# B&R Automation Studio project NAELD004C00R10L518F00 (part 19)

#### Act_OptP1031LifterMask.st
```iecst
ACTION Act_OptP1031LifterMask:

	// Interlock Power
	IF p_bLifterBtmAxisErr = TRUE AND p_bLifterBtmPwrOn = FALSE THEN
		fUIInRtStatOff(ADR(tyP1031MagSetTeach.tyMotionStdLifter.tyBtnPwr.uiMaskRtStat));
		tyP1031MagSetTeach.tyMotionStdLifter.tyBtnPwr.bValue		:= FALSE;
	ELSE
		fUIInRtStatHide(ADR(tyP1031MagSetTeach.tyMotionStdLifter.tyBtnPwr.uiMaskRtStat));
	END_IF

	// Interlock Others Move
	IF p_bLifterBtmAxisErr = TRUE OR p_bLifterBtmPwrOn = FALSE THEN
		fUIInRtStatOff(ADR(tyP1031MagSetTeach.tyMotionStdLifter.tyBtnOrigin.uiMaskRtStat));
		fUIInRtStatOff(ADR(tyP1031MagSetTeach.tyMotionStdLifter.tyBtnMovRel.uiMaskRtStat));
		fUIInRtStatOff(ADR(tyP1031MagSetTeach.tyMotionStdLifter.tyBtnJogUp.uiMaskRtStat));
		fUIInRtStatOff(ADR(tyP1031MagSetTeach.tyMotionStdLifter.tyBtnJogDown.uiMaskRtStat));
	ELSE
		fUIInRtStatHide(ADR(tyP1031MagSetTeach.tyMotionStdLifter.tyBtnOrigin.uiMaskRtStat));
		fUIInRtStatHide(ADR(tyP1031MagSetTeach.tyMotionStdLifter.tyBtnMovRel.uiMaskRtStat));
		fUIInRtStatHide(ADR(tyP1031MagSetTeach.tyMotionStdLifter.tyBtnJogUp.uiMaskRtStat));
		fUIInRtStatHide(ADR(tyP1031MagSetTeach.tyMotionStdLifter.tyBtnJogDown.uiMaskRtStat));
	END_IF

	// Interlock Move Absolute
	IF p_bLifterBtmAxisErr = TRUE OR p_bLifterBtmPwrOn = FALSE OR p_bLifterBtmIsHomed = FALSE THEN

		fUIInRtStatOff(ADR(tyP1031MagSetTeach.tyTeachLifterMag1Slt1Pos.tyBtn2.uiMaskRtStat));
		fUIInRtStatOff(ADR(tyP1031MagSetTeach.tyTeachLifterMag2Slt1Pos.tyBtn2.uiMaskRtStat));
		fUIInRtStatOff(ADR(tyP1031MagSetTeach.tyTeachLifterMag3Slt1Pos.tyBtn2.uiMaskRtStat));
		fUIInRtStatOff(ADR(tyP1031MagSetTeach.tyTeachLifterMag4Slt1Pos.tyBtn2.uiMaskRtStat));
		fUIInRtStatOff(ADR(tyP1031MagSetTeach.tyMotionStdLifter.tyBtnMovAbs.uiMaskRtStat));
	ELSE
		fUIInRtStatHide(ADR(tyP1031MagSetTeach.tyTeachLifterMag1Slt1Pos.tyBtn2.uiMaskRtStat));
		fUIInRtStatHide(ADR(tyP1031MagSetTeach.tyTeachLifterMag2Slt1Pos.tyBtn2.uiMaskRtStat));
		fUIInRtStatHide(ADR(tyP1031MagSetTeach.tyTeachLifterMag3Slt1Pos.tyBtn2.uiMaskRtStat));
		fUIInRtStatHide(ADR(tyP1031MagSetTeach.tyTeachLifterMag4Slt1Pos.tyBtn2.uiMaskRtStat));
		fUIInRtStatHide(ADR(tyP1031MagSetTeach.tyMotionStdLifter.tyBtnMovAbs.uiMaskRtStat));
	END_IF

	//Interlock Limit Sensor
	IF tyP1031MagSetTeach.tyMotionStdLifter.tyBtnDownLmtSen.bValue = TRUE THEN
		fUIInRtStatOff(ADR(tyP1031MagSetTeach.tyMotionStdLifter.tyBtnJogDown.uiMaskRtStat));
	END_IF

	IF tyP1031MagSetTeach.tyMotionStdLifter.tyBtnUpLmtSen.bValue = TRUE THEN
		fUIInRtStatOff(ADR(tyP1031MagSetTeach.tyMotionStdLifter.tyBtnJogUp.uiMaskRtStat));
	END_IF

	// Interlock When Moving
	IF tyP1031MagSetTeach.tyMotionStdLifter.tyBtnOrigin.bRtCompl = TRUE THEN
		fUIInRtStatOff(ADR(tyP1031MagSetTeach.tyMotionStdLifter.tyBtnMovAbs.uiMaskRtStat));
		fUIInRtStatOff(ADR(tyP1031MagSetTeach.tyMotionStdLifter.tyBtnMovRel.uiMaskRtStat));
		fUIInRtStatOff(ADR(tyP1031MagSetTeach.tyMotionStdLifter.tyBtnJogUp.uiMaskRtStat));
		fUIInRtStatOff(ADR(tyP1031MagSetTeach.tyMotionStdLifter.tyBtnJogDown.uiMaskRtStat));

		fUIInRtStatOff(ADR(tyP1031MagSetTeach.tyTeachLifterMag1Slt1Pos.tyBtn2.uiMaskRtStat));
		fUIInRtStatOff(ADR(tyP1031MagSetTeach.tyTeachLifterMag2Slt1Pos.tyBtn2.uiMaskRtStat));
		fUIInRtStatOff(ADR(tyP1031MagSetTeach.tyTeachLifterMag3Slt1Pos.tyBtn2.uiMaskRtStat));
		fUIInRtStatOff(ADR(tyP1031MagSetTeach.tyTeachLifterMag4Slt1Pos.tyBtn2.uiMaskRtStat));

	ELSIF tyP1031MagSetTeach.tyMotionStdLifter.tyBtnMovAbs.bRtCompl = TRUE THEN
		fUIInRtStatOff(ADR(tyP1031MagSetTeach.tyMotionStdLifter.tyBtnOrigin.uiMaskRtStat));
		fUIInRtStatOff(ADR(tyP1031MagSetTeach.tyMotionStdLifter.tyBtnMovRel.uiMaskRtStat));
		fUIInRtStatOff(ADR(tyP1031MagSetTeach.tyMotionStdLifter.tyBtnJogUp.uiMaskRtStat));
		fUIInRtStatOff(ADR(tyP1031MagSetTeach.tyMotionStdLifter.tyBtnJogDown.uiMaskRtStat));

		fUIInRtStatOff(ADR(tyP1031MagSetTeach.tyTeachLifterMag1Slt1Pos.tyBtn2.uiMaskRtStat));
		fUIInRtStatOff(ADR(tyP1031MagSetTeach.tyTeachLifterMag2Slt1Pos.tyBtn2.uiMaskRtStat));
		fUIInRtStatOff(ADR(tyP1031MagSetTeach.tyTeachLifterMag3Slt1Pos.tyBtn2.uiMaskRtStat));
		fUIInRtStatOff(ADR(tyP1031MagSetTeach.tyTeachLifterMag4Slt1Pos.tyBtn2.uiMaskRtStat));

	ELSIF tyP1031MagSetTeach.tyMotionStdLifter.tyBtnMovRel.bRtCompl = TRUE THEN
		fUIInRtStatOff(ADR(tyP1031MagSetTeach.tyMotionStdLifter.tyBtnOrigin.uiMaskRtStat));
		fUIInRtStatOff(ADR(tyP1031MagSetTeach.tyMotionStdLifter.tyBtnMovAbs.uiMaskRtStat));
		fUIInRtStatOff(ADR(tyP1031MagSetTeach.tyMotionStdLifter.tyBtnJogUp.uiMaskRtStat));
		fUIInRtStatOff(ADR(tyP1031MagSetTeach.tyMotionStdLifter.tyBtnJogDown.uiMaskRtStat));

		fUIInRtStatOff(ADR(tyP1031MagSetTeach.tyTeachLifterMag1Slt1Pos.tyBtn2.uiMaskRtStat));
		fUIInRtStatOff(ADR(tyP1031MagSetTeach.tyTeachLifterMag2Slt1Pos.tyBtn2.uiMaskRtStat));
		fUIInRtStatOff(ADR(tyP1031MagSetTeach.tyTeachLifterMag3Slt1Pos.tyBtn2.uiMaskRtStat));
		fUIInRtStatOff(ADR(tyP1031MagSetTeach.tyTeachLifterMag4Slt1Pos.tyBtn2.uiMaskRtStat));

	ELSIF tyP1031MagSetTeach.tyMotionStdLifter.tyBtnJogDown.bRtCompl = TRUE OR tyP1031MagSetTeach.tyMotionStdLifter.tyBtnJogDown.bValue = TRUE THEN
		fUIInRtStatOff(ADR(tyP1031MagSetTeach.tyMotionStdLifter.tyBtnOrigin.uiMaskRtStat));
		fUIInRtStatOff(ADR(tyP1031MagSetTeach.tyMotionStdLifter.tyBtnMovAbs.uiMaskRtStat));
		fUIInRtStatOff(ADR(tyP1031MagSetTeach.tyMotionStdLifter.tyBtnMovRel.uiMaskRtStat));
		fUIInRtStatOff(ADR(tyP1031MagSetTeach.tyMotionStdLifter.tyBtnJogUp.uiMaskRtStat));

		fUIInRtStatOff(ADR(tyP1031MagSetTeach.tyTeachLifterMag1Slt1Pos.tyBtn2.uiMaskRtStat));
		fUIInRtStatOff(ADR(tyP1031MagSetTeach.tyTeachLifterMag2Slt1Pos.tyBtn2.uiMaskRtStat));
		fUIInRtStatOff(ADR(tyP1031MagSetTeach.tyTeachLifterMag3Slt1Pos.tyBtn2.uiMaskRtStat));
		fUIInRtStatOff(ADR(tyP1031MagSetTeach.tyTeachLifterMag4Slt1Pos.tyBtn2.uiMaskRtStat));

	ELSIF tyP1031MagSetTeach.tyMotionStdLifter.tyBtnJogUp.bRtCompl = TRUE OR tyP1031MagSetTeach.tyMotionStdLifter.tyBtnJogUp.bValue = TRUE THEN
		fUIInRtStatOff(ADR(tyP1031MagSetTeach.tyMotionStdLifter.tyBtnOrigin.uiMaskRtStat));
		fUIInRtStatOff(ADR(tyP1031MagSetTeach.tyMotionStdLifter.tyBtnMovAbs.uiMaskRtStat));
		fUIInRtStatOff(ADR(tyP1031MagSetTeach.tyMotionStdLifter.tyBtnMovRel.uiMaskRtStat));
		fUIInRtStatOff(ADR(tyP1031MagSetTeach.tyMotionStdLifter.tyBtnJogDown.uiMaskRtStat));

		fUIInRtStatOff(ADR(tyP1031MagSetTeach.tyTeachLifterMag1Slt1Pos.tyBtn2.uiMaskRtStat));
		fUIInRtStatOff(ADR(tyP1031MagSetTeach.tyTeachLifterMag2Slt1Pos.tyBtn2.uiMaskRtStat));
		fUIInRtStatOff(ADR(tyP1031MagSetTeach.tyTeachLifterMag3Slt1Pos.tyBtn2.uiMaskRtStat));
		fUIInRtStatOff(ADR(tyP1031MagSetTeach.tyTeachLifterMag4Slt1Pos.tyBtn2.uiMaskRtStat));

	ELSIF tyP1031MagSetTeach.tyTeachLifterMag1Slt1Pos.tyBtn2.bRtCompl = TRUE THEN
		fUIInRtStatOff(ADR(tyP1031MagSetTeach.tyMotionStdLifter.tyBtnOrigin.uiMaskRtStat));
		fUIInRtStatOff(ADR(tyP1031MagSetTeach.tyMotionStdLifter.tyBtnMovAbs.uiMaskRtStat));
		fUIInRtStatOff(ADR(tyP1031MagSetTeach.tyMotionStdLifter.tyBtnMovRel.uiMaskRtStat));
		fUIInRtStatOff(ADR(tyP1031MagSetTeach.tyMotionStdLifter.tyBtnJogUp.uiMaskRtStat));
		fUIInRtStatOff(ADR(tyP1031MagSetTeach.tyMotionStdLifter.tyBtnJogDown.uiMaskRtStat));

	ELSIF tyP1031MagSetTeach.tyTeachLifterMag2Slt1Pos.tyBtn2.bRtCompl = TRUE THEN
		fUIInRtStatOff(ADR(tyP1031MagSetTeach.tyMotionStdLifter.tyBtnOrigin.uiMaskRtStat));
		fUIInRtStatOff(ADR(tyP1031MagSetTeach.tyMotionStdLifter.tyBtnMovAbs.uiMaskRtStat));
		fUIInRtStatOff(ADR(tyP1031MagSetTeach.tyMotionStdLifter.tyBtnMovRel.uiMaskRtStat));
		fUIInRtStatOff(ADR(tyP1031MagSetTeach.tyMotionStdLifter.tyBtnJogUp.uiMaskRtStat));
		fUIInRtStatOff(ADR(tyP1031MagSetTeach.tyMotionStdLifter.tyBtnJogDown.uiMaskRtStat));

	ELSIF tyP1031MagSetTeach.tyTeachLifterMag3Slt1Pos.tyBtn2.bRtCompl = TRUE THEN
		fUIInRtStatOff(ADR(tyP1031MagSetTeach.tyMotionStdLifter.tyBtnOrigin.uiMaskRtStat));
		fUIInRtStatOff(ADR(tyP1031MagSetTeach.tyMotionStdLifter.tyBtnMovAbs.uiMaskRtStat));
		fUIInRtStatOff(ADR(tyP1031MagSetTeach.tyMotionStdLifter.tyBtnMovRel.uiMaskRtStat));
		fUIInRtStatOff(ADR(tyP1031MagSetTeach.tyMotionStdLifter.tyBtnJogUp.uiMaskRtStat));
		fUIInRtStatOff(ADR(tyP1031MagSetTeach.tyMotionStdLifter.tyBtnJogDown.uiMaskRtStat));

	END_IF

	//Axis Error
	IF tyP1031MagSetTeach.tyMotionStdLifter.tyBtnPwr.bRtCompl = TRUE THEN
		fUIInRtStatOff(ADR(tyP1031MagSetTeach.tyMotionStdLifter.tyBtnRst.uiMaskRtStat));
	ELSE
		fUIInRtStatHide(ADR(tyP1031MagSetTeach.tyMotionStdLifter.tyBtnRst.uiMaskRtStat));
	END_IF

	//Interlock Button Get
	IF p_bLifterBtmAxisErr = TRUE OR p_bLifterBtmIsHomed = FALSE OR p_bLifterBtmFwdLmtSen = TRUE OR p_bLifterBtmRevLmtSen = TRUE THEN
		fUIInRtStatOff(ADR(tyP1031MagSetTeach.tyTeachLifterMag1Slt1Pos.tyBtn1.uiMaskRtStat));
		fUIInRtStatOff(ADR(tyP1031MagSetTeach.tyTeachLifterMag2Slt1Pos.tyBtn1.uiMaskRtStat));
		fUIInRtStatOff(ADR(tyP1031MagSetTeach.tyTeachLifterMag3Slt1Pos.tyBtn1.uiMaskRtStat));
		fUIInRtStatOff(ADR(tyP1031MagSetTeach.tyTeachLifterMag4Slt1Pos.tyBtn1.uiMaskRtStat));
	ELSE
		fUIInRtStatHide(ADR(tyP1031MagSetTeach.tyTeachLifterMag1Slt1Pos.tyBtn1.uiMaskRtStat));
		fUIInRtStatHide(ADR(tyP1031MagSetTeach.tyTeachLifterMag2Slt1Pos.tyBtn1.uiMaskRtStat));
		fUIInRtStatHide(ADR(tyP1031MagSetTeach.tyTeachLifterMag3Slt1Pos.tyBtn1.uiMaskRtStat));
		fUIInRtStatHide(ADR(tyP1031MagSetTeach.tyTeachLifterMag4Slt1Pos.tyBtn1.uiMaskRtStat));
	END_IF

END_ACTION
```

#### Act_OptP1031LifterUpdtDat.st
```iecst
ACTION Act_OptP1031LifterUpdtDat:

	tyP1031MagSetTeach.tyMotionStdLifter.tyNumCurrPos.diValue		:= p_diLifterBtmActualPos;
	tyP1031MagSetTeach.tyMotionStdLifter.tyNumErrCode.diValue		:= UDINT_TO_DINT(p_udiLifterBtmAxisErrID);
	tyP1031MagSetTeach.tyMotionStdLifter.tyBitmapPwr.usiValueIdx	:= BOOL_TO_USINT(p_bLifterBtmPwrOn);
	tyP1031MagSetTeach.tyMotionStdLifter.tyBitmapRst.usiValueIdx	:= BOOL_TO_USINT(NOT p_bLifterBtmAxisErr);
	tyP1031MagSetTeach.tyMotionStdLifter.tyBitmapOrigin.usiValueIdx	:= BOOL_TO_USINT(p_bLifterBtmIsHomed);
	tyP1031MagSetTeach.tyMotionStdLifter.tyBtnUpLmtSen.bValue		:= p_bLifterBtmUpSen;
	tyP1031MagSetTeach.tyMotionStdLifter.tyBtnDownLmtSen.bValue		:= p_bLifterBtmDownSen;

	//Machine Bitmap
	IF   (p_tyNtParamCurr.eProjMag = LDMagDual AND p_tyNtParamCurr.bMagAutoVerifyPrep = FALSE)
		OR (p_tyNtParamCurr.eProjMag = LDMagTriple AND p_tyNtParamCurr.bMagAutoVerifyPrep = FALSE)
		OR (p_tyNtParamCurr.eProjMag = LDMagDual AND p_tyNtParamCurr.bMagAutoVerifyPrep = TRUE)
		THEN
		IF p_bLifterBtmIsHomed = TRUE THEN

			IF p_diLifterBtmActualPos <= (p_tyNtParamCurr.tyUILifterTargetPos.diMax / 3) THEN
				tyP1031MagSetTeach.tyMotionStdLifter.tyBitmapMc.uiValueIdx 	:= 2;
			ELSIF p_diLifterBtmActualPos <= (p_tyNtParamCurr.tyUILifterTargetPos.diMax / 3 * 2) THEN
				tyP1031MagSetTeach.tyMotionStdLifter.tyBitmapMc.uiValueIdx 	:= 3;
			ELSE
				tyP1031MagSetTeach.tyMotionStdLifter.tyBitmapMc.uiValueIdx 	:= 4;
			END_IF

		ELSE
			tyP1031MagSetTeach.tyMotionStdLifter.tyBitmapMc.uiValueIdx	:= 2;
		END_IF

	ELSIF p_tyNtParamCurr.eProjMag = LDMagTriple AND p_tyNtParamCurr.bMagAutoVerifyPrep = TRUE
		THEN
		IF p_bLifterBtmIsHomed = TRUE THEN

			IF p_diLifterBtmActualPos <= (p_tyNtParamCurr.tyUILifterTargetPos.diMax / 3) THEN
				tyP1031MagSetTeach.tyMotionStdLifter.tyBitmapMc.uiValueIdx 	:= 23;
			ELSIF p_diLifterBtmActualPos <= (p_tyNtParamCurr.tyUILifterTargetPos.diMax / 3 * 2) THEN
				tyP1031MagSetTeach.tyMotionStdLifter.tyBitmapMc.uiValueIdx 	:= 24;
			ELSE
				tyP1031MagSetTeach.tyMotionStdLifter.tyBitmapMc.uiValueIdx 	:= 25;
			END_IF

		ELSE
			tyP1031MagSetTeach.tyMotionStdLifter.tyBitmapMc.uiValueIdx	:= 23;
		END_IF

	ELSIF p_tyNtParamCurr.eProjMag = LDMagQuadruple AND p_tyNtParamCurr.bMagAutoVerifyPrep = TRUE
		THEN
		IF p_bLifterBtmIsHomed = TRUE THEN

			IF p_diLifterBtmActualPos <= (p_tyNtParamCurr.tyUILifterTargetPos.diMax / 3) THEN
				tyP1031MagSetTeach.tyMotionStdLifter.tyBitmapMc.uiValueIdx 	:= 27;
			ELSIF p_diLifterBtmActualPos <= (p_tyNtParamCurr.tyUILifterTargetPos.diMax / 3 * 2) THEN
				tyP1031MagSetTeach.tyMotionStdLifter.tyBitmapMc.uiValueIdx 	:= 28;
			ELSE
				tyP1031MagSetTeach.tyMotionStdLifter.tyBitmapMc.uiValueIdx 	:= 29;
			END_IF

		ELSE
			tyP1031MagSetTeach.tyMotionStdLifter.tyBitmapMc.uiValueIdx	:= 27;
		END_IF
	END_IF

	IF p_tyNtParamCurr.eProjMag = LDMagTriple AND p_tyNtParamCurr.bProjLifterMagPlatform THEN
		IF 	tyP1031MagSetTeach.tyMotionStdLifter.tyBitmapMc.uiValueIdx < 400 THEN
			tyP1031MagSetTeach.tyMotionStdLifter.tyBitmapMc.uiValueIdx	:= tyP1031MagSetTeach.tyMotionStdLifter.tyBitmapMc.uiValueIdx + 400;
		END_IF
	ELSIF (p_tyNtParamCurr.eProjMag = LDMagDual OR p_tyNtParamCurr.eProjMag = LDMagTriple) AND p_tyNtParamCurr.bProjMotorizedPullerPrep = FALSE THEN
		IF 	tyP1031MagSetTeach.tyMotionStdLifter.tyBitmapMc.uiValueIdx < 200 THEN
			tyP1031MagSetTeach.tyMotionStdLifter.tyBitmapMc.uiValueIdx	:= tyP1031MagSetTeach.tyMotionStdLifter.tyBitmapMc.uiValueIdx + 200;
		END_IF
	ELSIF p_tyNtParamCurr.eProjMag = LDMagDual AND p_tyNtParamCurr.bProjMotorizedPullerPrep THEN
		IF p_tyNtParamCurr.sJobNo = '2023-0258A01' THEN
			tyP1031MagSetTeach.tyMotionStdLifter.tyBitmapMc.uiValueIdx	:= tyP1031MagSetTeach.tyMotionStdLifter.tyBitmapMc.uiValueIdx + 444-2;
		END_IF
	ELSIF p_tyNtParamCurr.eProjMag = LDMagTriple AND p_tyNtParamCurr.bMagAutoVerifyPrep = FALSE AND p_tyNtParamCurr.bProjMotorizedPullerPrep = TRUE
		THEN
		IF 	tyP1031MagSetTeach.tyMotionStdLifter.tyBitmapMc.uiValueIdx < 300 THEN
			tyP1031MagSetTeach.tyMotionStdLifter.tyBitmapMc.uiValueIdx	:= tyP1031MagSetTeach.tyMotionStdLifter.tyBitmapMc.uiValueIdx + 300;
		END_IF
	END_IF

END_ACTION
```

#### Act_OptP1031LifterKeypad.st
```iecst
ACTION Act_OptP1031LifterKeypad:

	IF fUIOutRtStatTPIsOpen(ADR(tyP1031MagSetTeach.tyMotionStdLifter.tyNumTargetPos.uiRtStat)) = TRUE THEN
		tyProperty.tyKeypad.tyStringTitle.sKeypadTitle		:= tyP1031MagSetTeach.tyMotionStdLifter.tyNumTargetPos.sKeypadTitle;

	ELSIF fUIOutRtStatTPIsOpen(ADR(tyP1026McSetTeach.tyMotionStdLifter.tyNumStepSize.uiRtStat)) = TRUE THEN
		tyProperty.tyKeypad.tyStringTitle.sKeypadTitle		:= tyP1031MagSetTeach.tyMotionStdLifter.tyNumStepSize.sKeypadTitle;

	ELSIF fUIOutRtStatTPIsOpen(ADR(tyP1031MagSetTeach.tyMotionStdLifter.tyNumNomSpd.uiRtStat)) = TRUE THEN
		tyProperty.tyKeypad.tyStringTitle.sKeypadTitle		:= tyP1031MagSetTeach.tyMotionStdLifter.tyNumNomSpd.sKeypadTitle;

	ELSIF fUIOutRtStatTPIsOpen(ADR(tyP1031MagSetTeach.tyMotionStdLifter.tyNumSlwSpd.uiRtStat)) = TRUE THEN
		tyProperty.tyKeypad.tyStringTitle.sKeypadTitle		:= tyP1031MagSetTeach.tyMotionStdLifter.tyNumSlwSpd.sKeypadTitle;

	ELSIF fUIOutRtStatTPIsOpen(ADR(tyP1031MagSetTeach.tyTeachLifterMag1Slt1Pos.tyNumNewSlt.uiRtStat)) = TRUE THEN
		tyProperty.tyKeypad.tyStringTitle.sKeypadTitle		:= tyP1031MagSetTeach.tyTeachLifterMag1Slt1Pos.tyNumNewSlt.sKeypadTitle;

	ELSIF fUIOutRtStatTPIsOpen(ADR(tyP1031MagSetTeach.tyTeachLifterMag2Slt1Pos.tyNumNewSlt.uiRtStat)) = TRUE THEN
		tyProperty.tyKeypad.tyStringTitle.sKeypadTitle		:= tyP1031MagSetTeach.tyTeachLifterMag2Slt1Pos.tyNumNewSlt.sKeypadTitle;

	ELSIF fUIOutRtStatTPIsOpen(ADR(tyP1031MagSetTeach.tyTeachLifterMag3Slt1Pos.tyNumNewSlt.uiRtStat)) = TRUE THEN
		tyProperty.tyKeypad.tyStringTitle.sKeypadTitle		:= tyP1031MagSetTeach.tyTeachLifterMag3Slt1Pos.tyNumNewSlt.sKeypadTitle;

	ELSIF fUIOutRtStatTPIsOpen(ADR(tyP1031MagSetTeach.tyTeachLifterMag4Slt1Pos.tyNumNewSlt.uiRtStat)) = TRUE THEN
		tyProperty.tyKeypad.tyStringTitle.sKeypadTitle		:= tyP1031MagSetTeach.tyTeachLifterMag4Slt1Pos.tyNumNewSlt.sKeypadTitle;

	END_IF

END_ACTION
```

#### Act_OptP1031LifterRstMnl.st
```iecst
ACTION Act_OptP1031LifterRstMnl:

	IF EDGEPOS((bManualMod = FALSE) OR (p_eLifterBtmStatus = Error)) THEN

		bJogSlow				:= FALSE;
		bJogFast				:= FALSE;
		fbJogSlowToFastDlyTm.IN	:= FALSE;

		tyP1031MagSetTeach.tyMotionStdLifter.tyBtnPwr.bRtCompl			:= FALSE;
		tyP1031MagSetTeach.tyMotionStdLifter.tyBtnStop.bRtCompl			:= FALSE;
		tyP1031MagSetTeach.tyMotionStdLifter.tyBtnOrigin.bRtCompl		:= FALSE;
		tyP1031MagSetTeach.tyMotionStdLifter.tyBtnRst.bRtCompl			:= FALSE;
		tyP1031MagSetTeach.tyMotionStdLifter.tyBtnMovAbs.bRtCompl		:= FALSE;
		tyP1031MagSetTeach.tyMotionStdLifter.tyBtnMovRel.bRtCompl		:= FALSE;
		tyP1031MagSetTeach.tyMotionStdLifter.tyBtnJogUp.bRtCompl		:= FALSE;
		tyP1031MagSetTeach.tyMotionStdLifter.tyBtnJogDown.bRtCompl		:= FALSE;

		tyP1031MagSetTeach.tyTeachLifterMag1Slt1Pos.tyBtn2.bRtCompl		:= FALSE;
		tyP1031MagSetTeach.tyTeachLifterMag2Slt1Pos.tyBtn2.bRtCompl		:= FALSE;
		tyP1031MagSetTeach.tyTeachLifterMag3Slt1Pos.tyBtn2.bRtCompl		:= FALSE;
		tyP1031MagSetTeach.tyTeachLifterMag4Slt1Pos.tyBtn2.bRtCompl		:= FALSE;

		tyP1031MagSetTeach.tyMotionStdLifter.tyBtnPwr.bValue			:= FALSE;
		tyP1031MagSetTeach.tyMotionStdLifter.tyBtnStop.bValue			:= TRUE;
		tyP1031MagSetTeach.tyMotionStdLifter.tyBtnOrigin.bValue			:= FALSE;
		tyP1031MagSetTeach.tyMotionStdLifter.tyBtnRst.bValue			:= FALSE;
		tyP1031MagSetTeach.tyMotionStdLifter.tyBtnMovAbs.bValue			:= FALSE;
		tyP1031MagSetTeach.tyMotionStdLifter.tyBtnMovRel.bValue			:= FALSE;
		tyP1031MagSetTeach.tyMotionStdLifter.tyBtnJogUp.bValue			:= FALSE;
		tyP1031MagSetTeach.tyMotionStdLifter.tyBtnJogDown.bValue		:= FALSE;

		tyP1031MagSetTeach.tyTeachLifterMag1Slt1Pos.tyBtn2.bValue		:= FALSE;
		tyP1031MagSetTeach.tyTeachLifterMag2Slt1Pos.tyBtn2.bValue		:= FALSE;
		tyP1031MagSetTeach.tyTeachLifterMag3Slt1Pos.tyBtn2.bValue		:= FALSE;
		tyP1031MagSetTeach.tyTeachLifterMag4Slt1Pos.tyBtn2.bValue		:= FALSE;

		tyP1031MagSetTeach.tyMotionStdLifter.tyBtnPwr.bRtLk				:= FALSE;
		tyP1031MagSetTeach.tyMotionStdLifter.tyBtnStop.bRtLk			:= TRUE;
		tyP1031MagSetTeach.tyMotionStdLifter.tyBtnOrigin.bRtLk			:= FALSE;
		tyP1031MagSetTeach.tyMotionStdLifter.tyBtnRst.bRtLk				:= FALSE;
		tyP1031MagSetTeach.tyMotionStdLifter.tyBtnMovAbs.bRtLk			:= FALSE;
		tyP1031MagSetTeach.tyMotionStdLifter.tyBtnMovRel.bRtLk			:= FALSE;
		tyP1031MagSetTeach.tyMotionStdLifter.tyBtnJogUp.bRtLk			:= FALSE;
		tyP1031MagSetTeach.tyMotionStdLifter.tyBtnJogDown.bRtLk			:= FALSE;

		tyP1031MagSetTeach.tyTeachLifterMag1Slt1Pos.tyBtn2.bRtLk		:= FALSE;
		tyP1031MagSetTeach.tyTeachLifterMag2Slt1Pos.tyBtn2.bRtLk		:= FALSE;
		tyP1031MagSetTeach.tyTeachLifterMag3Slt1Pos.tyBtn2.bRtLk		:= FALSE;
		tyP1031MagSetTeach.tyTeachLifterMag4Slt1Pos.tyBtn2.bRtLk		:= FALSE;

		tyP1031MagSetTeach.tyMotionStdLifter.tyBtnPwr.uiMaskRtStat		:= TRUE;
		tyP1031MagSetTeach.tyMotionStdLifter.tyBtnOrigin.uiMaskRtStat	:= FALSE;
		tyP1031MagSetTeach.tyMotionStdLifter.tyBtnRst.uiMaskRtStat		:= TRUE;
		tyP1031MagSetTeach.tyMotionStdLifter.tyBtnMovAbs.uiMaskRtStat	:= FALSE;
		tyP1031MagSetTeach.tyMotionStdLifter.tyBtnMovRel.uiMaskRtStat	:= FALSE;
		tyP1031MagSetTeach.tyMotionStdLifter.tyBtnJogUp.uiMaskRtStat	:= FALSE;
		tyP1031MagSetTeach.tyMotionStdLifter.tyBtnJogDown.uiMaskRtStat	:= FALSE;

		tyP1031MagSetTeach.tyTeachLifterMag1Slt1Pos.tyBtn2.uiMaskRtStat	:= FALSE;
		tyP1031MagSetTeach.tyTeachLifterMag2Slt1Pos.tyBtn2.uiMaskRtStat	:= FALSE;
		tyP1031MagSetTeach.tyTeachLifterMag3Slt1Pos.tyBtn2.uiMaskRtStat	:= FALSE;
		tyP1031MagSetTeach.tyTeachLifterMag4Slt1Pos.tyBtn2.uiMaskRtStat	:= FALSE;

		eInShutterAct	:= PneuActIdle;
		eOutShutterAct	:= PneuActIdle;
		eLifterBtmAct	:= LifterActIdle;

		tyP1031MagSetTeach.tyInOutletShutterFB.tyBtnClose.bRtCompl	:= FALSE;
		tyP1031MagSetTeach.tyInOutletShutterFB.tyBtnClose.bValue	:= FALSE;
		tyP1031MagSetTeach.tyInOutletShutterFB.tyBtnOpen.bRtCompl	:= FALSE;
		tyP1031MagSetTeach.tyInOutletShutterFB.tyBtnOpen.bValue	:= FALSE;
	END_IF

END_ACTION
```

#### Act_EntP1040Disp.st
```iecst
ACTION Act_EntP1040Disp:

	//Access Address
	p_tyC0005Main ACCESS ADR(tyCommon.tyMain);

	p_tyC0007Notif ACCESS ADR(tyCommon.tyNotif);

	p_tyC0008MsgBox ACCESS ADR(tyP1040ProdSet.tyMsgBoxHide);

	p_tyC0009Info ACCESS ADR(tyCommon.tyInfo);

	p_tyC0011RcpPopUp ACCESS ADR(tyP1040ProdSet.tyRcpPopUp);

	p_tyP1040ProdSet ACCESS ADR(tyP1040ProdSet.tyProdSet);
	tyP1040ProdSet.tyProdSet.tyStringSearch.sValue					:= '';

	//Display
	udiP1040SelectedRowOld	:= 0;

	tyP1040ProdSet.tyProdSet.tyBtnLongBrd.uiRtStat.0	:= NOT(p_tyNtParamCurr.bProjLongBrdPrep AND p_tyMcParamCurr.bLongBrdEn);

	//tyP1040ProdSet.tyProdSet.tyNumLastSlt.diValueMax	:= p_tyMagRcpCurrRcp.diTtlSlt;
	tyP1040ProdSet.tyProdSet.tyNumLastSlt.diValueMax	:= p_tyNtParamCurr.tyProdRcpMaxSlt.diMax;
	tyP1040ProdSet.tyProdSet.tyNumLastSltRear.diValueMax	:= p_tyMagRcpCurrRcp.diTtlSlt;

	fUIInRtStatHide(ADR(tyP1040ProdSet.tyRcpPopUp.tyLyr.uiRtStat));

END_ACTION
```

#### Act_OptP1040Del.st
```iecst
ACTION Act_OptP1040Del:

	IF tyP1040ProdSet.tyProdSet.tyBtnDelete.bRtCompl = TRUE THEN
		IF usiDelProdRcpStep = 0 THEN
			tyP1040ProdSet.tyProdSet.tyStringSearch.uiMaskRtStat				:= FALSE;
			tyP1040ProdSet.tyProdSet.tyTableRecipe.uiMaskRtStat					:= FALSE;

			IF tyP1040ProdSet.tyProdSet.tyTableRecipe.a_tyStringDataCol1[tyP1040Table.uiSelectedRow].sValue = p_tyProdRcpCurrRcp0.sRcpNm THEN
				p_tyC0008MsgBox ACCESS ADR(tyP1040ProdSet.tyMsgBoxDelCurrRcpAsk);

				IF tyP1040ProdSet.tyMsgBoxDelCurrRcpAsk.tyBtnNo.bRtCompl = TRUE THEN
					tyP1040ProdSet.tyMsgBoxDelCurrRcpAsk.tyBtnNo.bRtCompl 		:= FALSE;
					tyP1040ProdSet.tyMsgBoxDelCurrRcpAsk.tyBtnNo.bValue 		:= FALSE;

					p_tyC0008MsgBox ACCESS ADR(tyP1040ProdSet.tyMsgBoxHide);

					usiDelProdRcpStep	:= 99;
				END_IF
			ELSE
				p_tyC0008MsgBox ACCESS ADR(tyP1040ProdSet.tyMsgBoxDelAsk);

				IF tyP1040ProdSet.tyMsgBoxDelAsk.tyBtnYes.bRtCompl = TRUE THEN
					tyP1040ProdSet.tyMsgBoxDelAsk.tyBtnYes.bRtCompl				:= FALSE;
					tyP1040ProdSet.tyMsgBoxDelAsk.tyBtnYes.bValue				:= FALSE;

					p_tyC0008MsgBox ACCESS ADR(tyP1040ProdSet.tyMsgBoxHide);

					usiDelProdRcpStep	:= 1;

				ELSIF tyP1040ProdSet.tyMsgBoxDelAsk.tyBtnNo.bRtCompl = TRUE THEN
					tyP1040ProdSet.tyMsgBoxDelAsk.tyBtnNo.bRtCompl				:= FALSE;
					tyP1040ProdSet.tyMsgBoxDelAsk.tyBtnNo.bValue				:= FALSE;

					p_tyC0008MsgBox ACCESS ADR(tyP1040ProdSet.tyMsgBoxHide);

					usiDelProdRcpStep	:= 99;

				END_IF
			END_IF

		ELSIF usiDelProdRcpStep = 1 THEN
			tyProdRcpInfoIn.sRcpNm			:= tyP1040ProdSet.tyProdSet.tyTableRecipe.a_tyStringDataCol1[tyP1040Table.uiSelectedRow].sValue;

			eProdRcpAct					:= ProdRcpActDel;

			IF p_eProdRcpStat = ProdRcpActDel AND p_eProdRcpStatus = Done THEN
				eProdRcpAct				:= ProdRcpActIdle;

				IF p_bProdRcpNmEmpty = TRUE THEN
					usiDelProdRcpStep		:= 2;
				ELSIF p_bProdRcpNmNotExist = TRUE THEN
					usiDelProdRcpStep		:= 3;
				ELSE
					tyP1040ProdSet.tyProdSet.tyBtnSort.bValue := FALSE;
					tyP1040ProdSet.tyProdSet.tyStringSearch.sValue := '';

					bRefreshProdRcpTable	:= TRUE;
					bRefreshProdRcpDetail	:= TRUE;
					usiDelProdRcpStep		:= 99;
				END_IF

			ELSIF p_eProdRcpStatus = Error THEN
				p_tyC0008MsgBox ACCESS ADR(tyP1040ProdSet.tyMsgBoxDelErr);

				IF tyP1040ProdSet.tyMsgBoxDelErr.tyBtnNo.bRtCompl = TRUE THEN
					tyP1040ProdSet.tyMsgBoxDelErr.tyBtnNo.bRtCompl 				:= FALSE;
					tyP1040ProdSet.tyMsgBoxDelErr.tyBtnNo.bValue 				:= FALSE;

					p_tyC0008MsgBox ACCESS ADR(tyP1040ProdSet.tyMsgBoxHide);

					usiDelProdRcpStep		:= 99;
				END_IF
			END_IF

		ELSIF usiDelProdRcpStep = 2 THEN
			p_tyC0008MsgBox ACCESS ADR(tyP1040ProdSet.tyMsgBoxDelNmEmpty);

			IF tyP1040ProdSet.tyMsgBoxDelNmEmpty.tyBtnNo.bRtCompl = TRUE THEN
				tyP1040ProdSet.tyMsgBoxDelNmEmpty.tyBtnNo.bRtCompl 				:= FALSE;
				tyP1040ProdSet.tyMsgBoxDelNmEmpty.tyBtnNo.bValue 				:= FALSE;

				p_tyC0008MsgBox ACCESS ADR(tyP1040ProdSet.tyMsgBoxHide);

				usiDelProdRcpStep		:= 99;
			END_IF

		ELSIF usiDelProdRcpStep = 3 THEN
			p_tyC0008MsgBox ACCESS ADR(tyP1040ProdSet.tyMsgBoxDelNmNotExist);

			IF tyP1040ProdSet.tyMsgBoxDelNmNotExist.tyBtnNo.bRtCompl = TRUE THEN
				tyP1040ProdSet.tyMsgBoxDelNmNotExist.tyBtnNo.bRtCompl 		:= FALSE;
				tyP1040ProdSet.tyMsgBoxDelNmNotExist.tyBtnNo.bValue 		:= FALSE;

				p_tyC0008MsgBox ACCESS ADR(tyP1040ProdSet.tyMsgBoxHide);

				usiDelProdRcpStep	:= 99;
			END_IF

		ELSIF usiDelProdRcpStep = 99 THEN
			bRefreshProdRcpTable	:= FALSE;

			//Unmask
			tyP1040ProdSet.tyProdSet.tyStringSearch.uiMaskRtStat			:= TRUE;
			tyP1040ProdSet.tyProdSet.tyTableRecipe.uiMaskRtStat				:= TRUE;

			//Reset
			tyP1040ProdSet.tyProdSet.tyBtnDelete.bRtCompl					:= FALSE;
			tyP1040ProdSet.tyProdSet.tyBtnDelete.bValue						:= FALSE;

			usiDelProdRcpStep		:= 0;
		END_IF

	END_IF

END_ACTION
```

#### Act_OptP1040Keypad.st
```iecst
ACTION Act_OptP1040Keypad:

	tyP1040ProdSet.tyProdSet.tyNumFirstSlt.diValueMax	:= tyP1040ProdSet.tyProdSet.tyNumLastSlt.diValue;
	tyP1040ProdSet.tyProdSet.tyNumLastSlt.diValueMin	:= tyP1040ProdSet.tyProdSet.tyNumFirstSlt.diValue;
	tyP1040ProdSet.tyProdSet.tyNumPitch.diValueMax		:= tyP1040ProdSet.tyProdSet.tyNumLastSlt.diValue - tyP1040ProdSet.tyProdSet.tyNumFirstSlt.diValue + 1;

	tyP1040ProdSet.tyProdSet.tyNumFirstSltRear.diValueMax	:= tyP1040ProdSet.tyProdSet.tyNumLastSltRear.diValue;
	tyP1040ProdSet.tyProdSet.tyNumLastSltRear.diValueMin	:= tyP1040ProdSet.tyProdSet.tyNumFirstSltRear.diValue;
	tyP1040ProdSet.tyProdSet.tyNumPitchRear.diValueMax		:= tyP1040ProdSet.tyProdSet.tyNumLastSltRear.diValue - tyP1040ProdSet.tyProdSet.tyNumFirstSltRear.diValue + 1;

	IF fUIOutRtStatTPIsOpen(ADR(tyP1040ProdSet.tyProdSet.tyStringRecipeNm.uiRtStat)) THEN
		tyProperty.tyKeypad.tyStringTitle.sKeypadTitle	:= tyP1040ProdSet.tyProdSet.tyStringRecipeNm.sKeypadTitle;

	ELSIF fUIOutRtStatTPIsOpen(ADR(tyP1040ProdSet.tyProdSet.tyNumProdWidth.uiRtStat)) THEN
		IF p_tyNtParamCurr.bLFProdWidth2Prep THEN
			tyProperty.tyKeypad.tyStringTitle.sKeypadTitle	:= 'Product Width US';
		ELSE
			tyProperty.tyKeypad.tyStringTitle.sKeypadTitle	:= 'Product Width DS';
		END_IF

	ELSIF fUIOutRtStatTPIsOpen(ADR(tyP1040ProdSet.tyProdSet.tyNumProdWidth2.uiRtStat)) THEN
		tyProperty.tyKeypad.tyStringTitle.sKeypadTitle	:='Product Width DS';

	ELSIF fUIOutRtStatTPIsOpen(ADR(tyP1040ProdSet.tyProdSet.tyStringSearch.uiRtStat)) THEN
		tyProperty.tyKeypad.tyStringTitle.sKeypadTitle	:= tyP1040ProdSet.tyProdSet.tyStringSearch.sKeypadTitle;

	ELSIF fUIOutRtStatTPIsOpen(ADR(tyP1040ProdSet.tyProdSet.tyNumFirstSlt.uiRtStat)) THEN
		tyProperty.tyKeypad.tyStringTitle.sKeypadTitle	:= tyP1040ProdSet.tyProdSet.tyNumFirstSlt.sKeypadTitle;

	ELSIF fUIOutRtStatTPIsOpen(ADR(tyP1040ProdSet.tyProdSet.tyNumLastSlt.uiRtStat)) THEN
		tyProperty.tyKeypad.tyStringTitle.sKeypadTitle	:= tyP1040ProdSet.tyProdSet.tyNumLastSlt.sKeypadTitle;

	ELSIF fUIOutRtStatTPIsOpen(ADR(tyP1040ProdSet.tyProdSet.tyNumPitch.uiRtStat)) THEN
		tyProperty.tyKeypad.tyStringTitle.sKeypadTitle	:= tyP1040ProdSet.tyProdSet.tyNumPitch.sKeypadTitle;

	ELSIF fUIOutRtStatTPIsOpen(ADR(tyP1040ProdSet.tyProdSet.tyNumProdWidthRear.uiRtStat)) THEN
		tyProperty.tyKeypad.tyStringTitle.sKeypadTitle	:= tyP1040ProdSet.tyProdSet.tyNumProdWidth.sKeypadTitle;

	ELSIF fUIOutRtStatTPIsOpen(ADR(tyP1040ProdSet.tyProdSet.tyNumPitchRear.uiRtStat)) THEN
		tyProperty.tyKeypad.tyStringTitle.sKeypadTitle	:= tyP1040ProdSet.tyProdSet.tyNumPitch.sKeypadTitle;

	ELSIF fUIOutRtStatTPIsOpen(ADR(tyP1040ProdSet.tyProdSet.tyNumFirstSltRear.uiRtStat)) THEN
		tyProperty.tyKeypad.tyStringTitle.sKeypadTitle	:= tyP1040ProdSet.tyProdSet.tyNumFirstSlt.sKeypadTitle;

	ELSIF fUIOutRtStatTPIsOpen(ADR(tyP1040ProdSet.tyProdSet.tyNumLastSltRear.uiRtStat)) THEN
		tyProperty.tyKeypad.tyStringTitle.sKeypadTitle	:= tyP1040ProdSet.tyProdSet.tyNumLastSlt.sKeypadTitle;

	ELSIF fUIOutRtStatTPIsOpen(ADR(tyP1040ProdSet.tyProdSet.tyNumPshrOffset.uiRtStat))THEN
		tyProperty.tyKeypad.tyStringTitle.sKeypadTitle	:= tyP1040ProdSet.tyProdSet.tyNumPshrOffset.sKeypadTitle;

	ELSE
		tyProperty.tyKeypad.tyStringTitle.sKeypadTitle	:= '';

	END_IF

END_ACTION
```

#### Act_OptP1040Limit.st
```iecst
ACTION Act_OptP1040Limit:
//pulller closing ref
//	IF tyP1040ProdSet.tyProdSet.tyBtnSort.bValue THEN //sorted == by name
//		IF tyP1040ProdSet.tyProdSet.tyNumPshrOffset.diValueMin<0 THEN
//			tyP1040ProdSet.tyProdSet.tyNumPshrOffset.diValueMin		:= -(tyP1040ProdSet.tyProdSet.tyNumProdWidth.diValue/2-p_tyMcParamCurr.diAWPusherAtHmPosInUM );
//		ELSE
//			tyP1040ProdSet.tyProdSet.tyNumPshrOffset.diValueMin		:=0;
//		END_IF
//
//		tyP1040ProdSet.tyProdSet.tyNumPshrOffset.diValueMax		:= (tyP1040ProdSet.tyProdSet.tyNumProdWidth.diValue/2-p_tyMcParamCurr.diAWPusherAtHmPosInUM-5000 );
//	ELSE // by default == curr list
//		IF tyP1040ProdSet.tyProdSet.tyNumPshrOffset.diValueMin<0 THEN
			tyP1040ProdSet.tyProdSet.tyNumPshrOffset.diValueMin		:= -(tyP1040ProdSet.tyProdSet.tyNumProdWidth.diValue/2-50000);
//		ELSE
//			tyP1040ProdSet.tyProdSet.tyNumPshrOffset.diValueMin		:=0;
//		END_IF

//		tyP1040ProdSet.tyProdSet.tyNumPshrOffset.diValueMax		:= (tyP1040ProdSet.tyProdSet.tyNumProdWidth.diValue/2-p_tyMcParamCurr.diAWPusherAtHmPosInUM-5000 );
		tyP1040ProdSet.tyProdSet.tyNumPshrOffset.diValueMax		:= (tyP1040ProdSet.tyProdSet.tyNumProdWidth.diValue/2-50000 );
//	END_IF

END_ACTION
```

#### Act_OptP1040LoadData.st
```iecst
ACTION Act_OptP1040LoadData:

	udiP1040SelectedRow		:= STRING_TO_UDINT(tyP1040ProdSet.tyProdSet.tyTableRecipe.a_tyStringDataCol0[tyP1040Table.uiSelectedRow].sValue);

	IF udiP1040SelectedRow <> udiP1040SelectedRowOld OR bRefreshProdRcpDetail = TRUE OR bUpdateP1040LoadData THEN
		IF tyP1040ProdSet.tyProdSet.tyStringSearch.sValue = '' THEN
			IF tyP1040ProdSet.tyProdSet.tyTableRecipe.a_tyStringDataCol1[tyP1040Table.uiSelectedRow].sValue <> '' THEN
				//Update Recipe Data
				IF tyP1040ProdSet.tyProdSet.tyBtnSort.bValue THEN
					tyP1040ProdSet.tyProdSet.tyStringRecipeNm.sValue		:= p_tyProdRcpSortedList[udiP1040SelectedRow].sRcpNm;
					tyP1040ProdSet.tyProdSet.tyNumProdWidth.diValue			:= p_tyProdRcpSortedList[udiP1040SelectedRow].diWidthInUM;
					tyP1040ProdSet.tyProdSet.tyNumProdWidth2.diValue		:= p_tyProdRcpSortedList[udiP1040SelectedRow].diWidthInUM2;
					tyP1040ProdSet.tyProdSet.tyNumLastSlt.diValue			:= p_tyProdRcpSortedList[udiP1040SelectedRow].diMaxSltValue;
					tyP1040ProdSet.tyProdSet.tyNumFirstSlt.diValue			:= p_tyProdRcpSortedList[udiP1040SelectedRow].diMinSltValue;
					tyP1040ProdSet.tyProdSet.tyNumPitch.diValue				:= p_tyProdRcpSortedList[udiP1040SelectedRow].diPitch;
					tyP1040ProdSet.tyProdSet.tyDrpDnMcMode.usiValueIdx		:= p_tyProdRcpSortedList[udiP1040SelectedRow].usiMcMod;
					tyP1040ProdSet.tyProdSet.tyDrpDnFlippedBrd.usiValueIdx	:= p_tyProdRcpSortedList[udiP1040SelectedRow].usiFlippedBrd;
					tyP1040ProdSet.tyProdSet.tyBtnToptoBtm.bValue			:= p_tyProdRcpSortedList[udiP1040SelectedRow].bTopToBtm;
					tyP1040ProdSet.tyProdSet.tyBtnLongBrd.bValue			:= p_tyProdRcpSortedList[udiP1040SelectedRow].bLongBrd;

					tyP1040ProdSet.tyProdSet.tyNumProdWidthRear.diValue		:= p_tyProdRcpSortedList[udiP1040SelectedRow].diWidthInUMRear;
					tyP1040ProdSet.tyProdSet.tyNumLastSltRear.diValue		:= p_tyProdRcpSortedList[udiP1040SelectedRow].diMaxSltValueRear;
					tyP1040ProdSet.tyProdSet.tyNumFirstSltRear.diValue		:= p_tyProdRcpSortedList[udiP1040SelectedRow].diMinSltValueRear;
					tyP1040ProdSet.tyProdSet.tyNumPitchRear.diValue			:= p_tyProdRcpSortedList[udiP1040SelectedRow].diPitchRear;
					tyP1040ProdSet.tyProdSet.tyNumMtrPshrExtSpd.diValue		:= p_tyProdRcpSortedList[udiP1040SelectedRow].diMtrPshrExtSpd;
					tyP1040ProdSet.tyProdSet.tyNumMtrPshrExtTorq.diValue	:= p_tyProdRcpSortedList[udiP1040SelectedRow].diMtrPshrExtTorq;
					tyP1040ProdSet.tyProdSet.tyNumPshrOffset.diValue		:= p_tyProdRcpSortedList[udiP1040SelectedRow].diPshrOffset;
				ELSE
					tyP1040ProdSet.tyProdSet.tyStringRecipeNm.sValue		:= p_tyProdRcpCurrList[udiP1040SelectedRow].sRcpNm;
					tyP1040ProdSet.tyProdSet.tyNumProdWidth.diValue			:= p_tyProdRcpCurrList[udiP1040SelectedRow].diWidthInUM;
					tyP1040ProdSet.tyProdSet.tyNumProdWidth2.diValue		:= p_tyProdRcpCurrList[udiP1040SelectedRow].diWidthInUM2;
					tyP1040ProdSet.tyProdSet.tyNumLastSlt.diValue			:= p_tyProdRcpCurrList[udiP1040SelectedRow].diMaxSltValue;
					tyP1040ProdSet.tyProdSet.tyNumFirstSlt.diValue			:= p_tyProdRcpCurrList[udiP1040SelectedRow].diMinSltValue;
					tyP1040ProdSet.tyProdSet.tyNumPitch.diValue				:= p_tyProdRcpCurrList[udiP1040SelectedRow].diPitch;
					tyP1040ProdSet.tyProdSet.tyDrpDnMcMode.usiValueIdx		:= p_tyProdRcpCurrList[udiP1040SelectedRow].usiMcMod;
					tyP1040ProdSet.tyProdSet.tyDrpDnFlippedBrd.usiValueIdx	:= p_tyProdRcpCurrList[udiP1040SelectedRow].usiFlippedBrd;
					tyP1040ProdSet.tyProdSet.tyBtnToptoBtm.bValue			:= p_tyProdRcpCurrList[udiP1040SelectedRow].bTopToBtm;
					tyP1040ProdSet.tyProdSet.tyBtnLongBrd.bValue			:= p_tyProdRcpCurrList[udiP1040SelectedRow].bLongBrd;

					tyP1040ProdSet.tyProdSet.tyNumProdWidthRear.diValue		:= p_tyProdRcpCurrList[udiP1040SelectedRow].diWidthInUMRear;
					tyP1040ProdSet.tyProdSet.tyNumLastSltRear.diValue		:= p_tyProdRcpCurrList[udiP1040SelectedRow].diMaxSltValueRear;
					tyP1040ProdSet.tyProdSet.tyNumFirstSltRear.diValue		:= p_tyProdRcpCurrList[udiP1040SelectedRow].diMinSltValueRear;
					tyP1040ProdSet.tyProdSet.tyNumPitchRear.diValue			:= p_tyProdRcpCurrList[udiP1040SelectedRow].diPitchRear;
					tyP1040ProdSet.tyProdSet.tyNumMtrPshrExtSpd.diValue		:= p_tyProdRcpCurrList[udiP1040SelectedRow].diMtrPshrExtSpd;
					tyP1040ProdSet.tyProdSet.tyNumMtrPshrExtTorq.diValue	:= p_tyProdRcpCurrList[udiP1040SelectedRow].diMtrPshrExtTorq;
					tyP1040ProdSet.tyProdSet.tyNumPshrOffset.diValue		:= p_tyProdRcpCurrList[udiP1040SelectedRow].diPshrOffset;
				END_IF
			ELSE
				tyP1040ProdSet.tyProdSet.tyStringRecipeNm.sValue		:= '';
				tyP1040ProdSet.tyProdSet.tyNumProdWidth.diValue			:= 100000;
				tyP1040ProdSet.tyProdSet.tyNumProdWidth2.diValue		:= 100000;
				tyP1040ProdSet.tyProdSet.tyNumLastSlt.diValue			:= p_tyNtParamCurr.tyProdRcpMaxSlt.diMax;//p_tyMagRcpCurrRcp.diTtlSlt;
				tyP1040ProdSet.tyProdSet.tyNumFirstSlt.diValue			:= p_tyNtParamCurr.diProjMagMinSlt;
				tyP1040ProdSet.tyProdSet.tyNumPitch.diValue				:= 1;
				tyP1040ProdSet.tyProdSet.tyDrpDnMcMode.usiValueIdx		:= p_tyMcParamCurr.usiDefaultMcMod;
				tyP1040ProdSet.tyProdSet.tyDrpDnFlippedBrd.usiValueIdx	:= p_tyMcParamCurr.usiDefaultFlippedBrd;
				tyP1040ProdSet.tyProdSet.tyBtnToptoBtm.bValue			:= p_tyNtParamCurr.bProjTopToBtmDefault;
				tyP1040ProdSet.tyProdSet.tyBtnLongBrd.bValue			:= FALSE;

				tyP1040ProdSet.tyProdSet.tyNumProdWidthRear.diValue		:= 100000;
				tyP1040ProdSet.tyProdSet.tyNumPitchRear.diValue			:= 1;
				tyP1040ProdSet.tyProdSet.tyNumLastSltRear.diValue		:= p_tyMagRcpCurrRcp.diTtlSlt;
				tyP1040ProdSet.tyProdSet.tyNumFirstSltRear.diValue		:= p_tyNtParamCurr.diProjMagMinSlt;
				tyP1040ProdSet.tyProdSet.tyNumMtrPshrExtSpd.diValue		:= p_tyNtParamCurr.tyProdRcpMtrPshrExtSpd.diMax-1;
				tyP1040ProdSet.tyProdSet.tyNumMtrPshrExtTorq.diValue	:= p_tyNtParamCurr.tyProdRcpMtrPshrExtTorq.diMin+50;
				tyP1040ProdSet.tyProdSet.tyNumPshrOffset.diValue		:= 0;

			END_IF

		ELSE

			IF tyP1040ProdSet.tyProdSet.tyTableRecipe.a_tyStringDataCol1[tyP1040Table.uiSelectedRow].sValue <> '' THEN
				//Update Recipe Data
				IF tyP1040ProdSet.tyProdSet.tyBtnSort.bValue THEN
					tyP1040ProdSet.tyProdSet.tyStringRecipeNm.sValue		:= p_tyProdRcpSortedList[udiP1040SelectedRow].sRcpNm;
					tyP1040ProdSet.tyProdSet.tyNumProdWidth.diValue			:= p_tyProdRcpSortedList[udiP1040SelectedRow].diWidthInUM;
					tyP1040ProdSet.tyProdSet.tyNumProdWidth2.diValue		:= p_tyProdRcpSortedList[udiP1040SelectedRow].diWidthInUM2;
					tyP1040ProdSet.tyProdSet.tyNumLastSlt.diValue			:= p_tyProdRcpSortedList[udiP1040SelectedRow].diMaxSltValue;
					tyP1040ProdSet.tyProdSet.tyNumFirstSlt.diValue			:= p_tyProdRcpSortedList[udiP1040SelectedRow].diMinSltValue;
					tyP1040ProdSet.tyProdSet.tyNumPitch.diValue				:= p_tyProdRcpSortedList[udiP1040SelectedRow].diPitch;
					tyP1040ProdSet.tyProdSet.tyDrpDnMcMode.usiValueIdx		:= p_tyProdRcpSortedList[udiP1040SelectedRow].usiMcMod;
					tyP1040ProdSet.tyProdSet.tyDrpDnFlippedBrd.usiValueIdx	:= p_tyProdRcpSortedList[udiP1040SelectedRow].usiFlippedBrd;
					tyP1040ProdSet.tyProdSet.tyBtnToptoBtm.bValue			:= p_tyProdRcpSortedList[udiP1040SelectedRow].bTopToBtm;
					tyP1040ProdSet.tyProdSet.tyBtnLongBrd.bValue			:= p_tyProdRcpSortedList[udiP1040SelectedRow].bLongBrd;

					tyP1040ProdSet.tyProdSet.tyNumProdWidthRear.diValue		:= p_tyProdRcpSortedList[udiP1040SelectedRow].diWidthInUMRear;
					tyP1040ProdSet.tyProdSet.tyNumLastSltRear.diValue		:= p_tyProdRcpSortedList[udiP1040SelectedRow].diMaxSltValueRear;
					tyP1040ProdSet.tyProdSet.tyNumFirstSltRear.diValue		:= p_tyProdRcpSortedList[udiP1040SelectedRow].diMinSltValueRear;
					tyP1040ProdSet.tyProdSet.tyNumPitchRear.diValue			:= p_tyProdRcpSortedList[udiP1040SelectedRow].diPitchRear;
					tyP1040ProdSet.tyProdSet.tyNumMtrPshrExtSpd.diValue		:= p_tyProdRcpSortedList[udiP1040SelectedRow].diMtrPshrExtSpd;
					tyP1040ProdSet.tyProdSet.tyNumMtrPshrExtTorq.diValue	:= p_tyProdRcpSortedList[udiP1040SelectedRow].diMtrPshrExtTorq;
					tyP1040ProdSet.tyProdSet.tyNumPshrOffset.diValue		:= p_tyProdRcpSortedList[udiP1040SelectedRow].diPshrOffset;
				ELSE
					tyP1040ProdSet.tyProdSet.tyStringRecipeNm.sValue		:= p_tyProdRcpFilterList[udiP1040SelectedRow].sRcpNm;
					tyP1040ProdSet.tyProdSet.tyNumProdWidth.diValue			:= p_tyProdRcpFilterList[udiP1040SelectedRow].diWidthInUM;
					tyP1040ProdSet.tyProdSet.tyNumProdWidth2.diValue		:= p_tyProdRcpFilterList[udiP1040SelectedRow].diWidthInUM2;
					tyP1040ProdSet.tyProdSet.tyNumProdWidthRear.diValue		:= p_tyProdRcpFilterList[udiP1040SelectedRow].diWidthInUMRear;
					tyP1040ProdSet.tyProdSet.tyNumLastSlt.diValue			:= p_tyProdRcpFilterList[udiP1040SelectedRow].diMaxSltValue;
					tyP1040ProdSet.tyProdSet.tyNumFirstSlt.diValue			:= p_tyProdRcpFilterList[udiP1040SelectedRow].diMinSltValue;
					tyP1040ProdSet.tyProdSet.tyNumPitch.diValue				:= p_tyProdRcpFilterList[udiP1040SelectedRow].diPitch;
					tyP1040ProdSet.tyProdSet.tyDrpDnMcMode.usiValueIdx		:= p_tyProdRcpFilterList[udiP1040SelectedRow].usiMcMod;
					tyP1040ProdSet.tyProdSet.tyDrpDnFlippedBrd.usiValueIdx	:= p_tyProdRcpFilterList[udiP1040SelectedRow].usiFlippedBrd;
					tyP1040ProdSet.tyProdSet.tyBtnToptoBtm.bValue			:= p_tyProdRcpFilterList[udiP1040SelectedRow].bTopToBtm;
					tyP1040ProdSet.tyProdSet.tyBtnLongBrd.bValue			:= p_tyProdRcpFilterList[udiP1040SelectedRow].bLongBrd;

					tyP1040ProdSet.tyProdSet.tyNumProdWidthRear.diValue		:= p_tyProdRcpFilterList[udiP1040SelectedRow].diWidthInUMRear;
					tyP1040ProdSet.tyProdSet.tyNumLastSltRear.diValue		:= p_tyProdRcpFilterList[udiP1040SelectedRow].diMaxSltValueRear;
					tyP1040ProdSet.tyProdSet.tyNumFirstSltRear.diValue		:= p_tyProdRcpFilterList[udiP1040SelectedRow].diMinSltValueRear;
					tyP1040ProdSet.tyProdSet.tyNumPitchRear.diValue			:= p_tyProdRcpFilterList[udiP1040SelectedRow].diPitchRear;
					tyP1040ProdSet.tyProdSet.tyNumMtrPshrExtSpd.diValue		:= p_tyProdRcpFilterList[udiP1040SelectedRow].diMtrPshrExtSpd;
					tyP1040ProdSet.tyProdSet.tyNumMtrPshrExtTorq.diValue	:= p_tyProdRcpFilterList[udiP1040SelectedRow].diMtrPshrExtTorq;
					tyP1040ProdSet.tyProdSet.tyNumPshrOffset.diValue		:= p_tyProdRcpFilterList[udiP1040SelectedRow].diPshrOffset;
				END_IF
			ELSE
				tyP1040ProdSet.tyProdSet.tyStringRecipeNm.sValue		:= '';
				tyP1040ProdSet.tyProdSet.tyNumProdWidth.diValue			:= 100000;
				tyP1040ProdSet.tyProdSet.tyNumProdWidth2.diValue		:= 100000;
				tyP1040ProdSet.tyProdSet.tyNumLastSlt.diValue			:= p_tyNtParamCurr.tyProdRcpMaxSlt.diMax;//p_tyMagRcpCurrRcp.diTtlSlt;
				tyP1040ProdSet.tyProdSet.tyNumFirstSlt.diValue			:= p_tyNtParamCurr.diProjMagMinSlt;
				tyP1040ProdSet.tyProdSet.tyNumPitch.diValue				:= 1;
				tyP1040ProdSet.tyProdSet.tyDrpDnMcMode.usiValueIdx		:= p_tyMcParamCurr.usiDefaultMcMod;
				tyP1040ProdSet.tyProdSet.tyDrpDnFlippedBrd.usiValueIdx	:= p_tyMcParamCurr.usiDefaultFlippedBrd;
				tyP1040ProdSet.tyProdSet.tyBtnToptoBtm.bValue			:= p_tyNtParamCurr.bProjTopToBtmDefault;
				tyP1040ProdSet.tyProdSet.tyBtnLongBrd.bValue			:= FALSE;

				tyP1040ProdSet.tyProdSet.tyNumProdWidthRear.diValue		:= 100000;
				tyP1040ProdSet.tyProdSet.tyNumLastSltRear.diValue		:= p_tyMagRcpCurrRcp.diTtlSlt;
				tyP1040ProdSet.tyProdSet.tyNumFirstSltRear.diValue		:= p_tyNtParamCurr.diProjMagMinSlt;
				tyP1040ProdSet.tyProdSet.tyNumPitchRear.diValue			:= 1;
				tyP1040ProdSet.tyProdSet.tyNumMtrPshrExtSpd.diValue		:= p_tyNtParamCurr.tyProdRcpMtrPshrExtSpd.diMax-1;
				tyP1040ProdSet.tyProdSet.tyNumMtrPshrExtTorq.diValue	:= p_tyNtParamCurr.tyProdRcpMtrPshrExtTorq.diMin+50;
				tyP1040ProdSet.tyProdSet.tyNumPshrOffset.diValue		:= 0;
			END_IF

		END_IF

		bUpdateP1040LoadData 		:= FALSE;
		bRefreshProdRcpDetail		:= FALSE;
		udiP1040SelectedRowOld 		:= udiP1040SelectedRow;

		fUIInRtStatOff(ADR(tyP1040ProdSet.tyProdSet.tyBtnSave.uiMaskRtStat));

	END_IF

END_ACTION
```

#### Act_OptP1040Mask.st
```iecst
ACTION Act_OptP1040Mask:

	IF tyP1040ProdSet.tyProdSet.tyStringRecipeNm.bRtCompl		OR tyP1040ProdSet.tyProdSet.tyNumProdWidth.bRtCompl
		OR tyP1040ProdSet.tyProdSet.tyNumFirstSlt.bRtCompl		OR tyP1040ProdSet.tyProdSet.tyNumLastSlt.bRtCompl
		OR tyP1040ProdSet.tyProdSet.tyNumPitch.bRtCompl			OR tyP1040ProdSet.tyProdSet.tyDrpDnMcMode.bRtCompl
		OR tyP1040ProdSet.tyProdSet.tyDrpDnFlippedBrd.bRtCompl	OR tyP1040ProdSet.tyProdSet.tyBtnToptoBtm.bRtCompl
		OR tyP1040ProdSet.tyProdSet.tyBtnLongBrd.bRtCompl 		OR tyP1040ProdSet.tyProdSet.tyNumProdWidth2.bRtCompl
		OR tyP1040ProdSet.tyProdSet.tyNumProdWidthRear.bRtCompl OR tyP1040ProdSet.tyProdSet.tyNumPitchRear.bRtCompl
		OR tyP1040ProdSet.tyProdSet.tyNumFirstSltRear.bRtCompl  OR tyP1040ProdSet.tyProdSet.tyNumLastSltRear.bRtCompl
		OR tyP1040ProdSet.tyProdSet.tyNumMtrPshrExtSpd.bRtCompl OR tyP1040ProdSet.tyProdSet.tyNumMtrPshrExtTorq.bRtCompl
		OR tyP1040ProdSet.tyProdSet.tyNumPshrOffset.bRtCompl
		THEN

		fUIInRtStatHide(ADR(tyP1040ProdSet.tyProdSet.tyBtnSave.uiMaskRtStat));

		tyP1040ProdSet.tyProdSet.tyStringRecipeNm.bRtCompl	:= FALSE;
		tyP1040ProdSet.tyProdSet.tyNumProdWidth.bRtCompl	:= FALSE;
		tyP1040ProdSet.tyProdSet.tyNumProdWidth2.bRtCompl	:= FALSE;
		tyP1040ProdSet.tyProdSet.tyNumFirstSlt.bRtCompl		:= FALSE;
		tyP1040ProdSet.tyProdSet.tyNumLastSlt.bRtCompl		:= FALSE;
		tyP1040ProdSet.tyProdSet.tyNumPitch.bRtCompl		:= FALSE;
		tyP1040ProdSet.tyProdSet.tyDrpDnMcMode.bRtCompl		:= FALSE;
		tyP1040ProdSet.tyProdSet.tyDrpDnFlippedBrd.bRtCompl	:= FALSE;
		tyP1040ProdSet.tyProdSet.tyBtnToptoBtm.bRtCompl		:= FALSE;
		tyP1040ProdSet.tyProdSet.tyBtnLongBrd.bRtCompl		:= FALSE;
		tyP1040ProdSet.tyProdSet.tyNumProdWidthRear.bRtCompl:= FALSE;

		tyP1040ProdSet.tyProdSet.tyNumProdWidthRear.bRtCompl:= FALSE;
		tyP1040ProdSet.tyProdSet.tyNumPitchRear.bRtCompl	:= FALSE;
		tyP1040ProdSet.tyProdSet.tyNumFirstSltRear.bRtCompl	:= FALSE;
		tyP1040ProdSet.tyProdSet.tyNumLastSltRear.bRtCompl	:= FALSE;
		tyP1040ProdSet.tyProdSet.tyNumMtrPshrExtSpd.bRtCompl	:= FALSE;
		tyP1040ProdSet.tyProdSet.tyNumMtrPshrExtTorq.bRtCompl	:= FALSE;
		tyP1040ProdSet.tyProdSet.tyNumPshrOffset.bRtCompl		:= FALSE;
	END_IF

	IF (tyP1040ProdSet.tyProdSet.tyTableRecipe.a_tyStringDataCol1[tyP1040Table.uiSelectedRow].sValue <> '') AND (tyP1040ProdSet.tyProdSet.tyBtnSave.bRtCompl = FALSE) AND (tyP1040ProdSet.tyProdSet.tyBtnToXML.bRtCompl = FALSE) AND (tyP1040ProdSet.tyProdSet.tyBtnFromXML.bRtCompl = FALSE) THEN
		fUIInRtStatHide(ADR(tyP1040ProdSet.tyProdSet.tyBtnDelete.uiMaskRtStat));
	ELSE
		fUIInRtStatOff(ADR(tyP1040ProdSet.tyProdSet.tyBtnDelete.uiMaskRtStat));
	END_IF

	tyP1040ProdSet.tyProdSet.tyBtnToXML.uiMaskRtStat.0		:= (tyP1040ProdSet.tyProdSet.tyBtnSave.uiMaskRtStat.0 = FALSE) AND (tyP1040ProdSet.tyProdSet.tyBtnDelete.bRtCompl = FALSE) AND (tyP1040ProdSet.tyProdSet.tyBtnFromXML.bRtCompl = FALSE);
	tyP1040ProdSet.tyProdSet.tyBtnFromXML.uiMaskRtStat.0	:= (tyP1040ProdSet.tyProdSet.tyBtnSave.uiMaskRtStat.0 = FALSE) AND (tyP1040ProdSet.tyProdSet.tyBtnDelete.bRtCompl = FALSE) AND (tyP1040ProdSet.tyProdSet.tyBtnToXML.bRtCompl = FALSE);

	tyP1040ProdSet.tyProdSet.tyBtnSort.uiMaskRtStat.0		:= (tyP1040ProdSet.tyProdSet.tyTableRecipe.a_tyStringDataCol1[1].sValue <> '') AND (tyP1040ProdSet.tyProdSet.tyStringSearch.bRtCompl = FALSE)
																AND (tyP1040ProdSet.tyProdSet.tyBtnSave.uiMaskRtStat.0 = FALSE) AND (tyP1040ProdSet.tyProdSet.tyBtnDelete.bRtCompl = FALSE)
																AND (tyP1040ProdSet.tyProdSet.tyBtnToXML.bRtCompl = FALSE) AND (tyP1040ProdSet.tyProdSet.tyBtnFromXML.bRtCompl = FALSE);

END_ACTION
```

#### Act_OptP1040Save.st
```iecst
ACTION Act_OptP1040Save:

	IF tyP1040ProdSet.tyProdSet.tyBtnSave.bRtCompl = TRUE THEN
		IF usiSaveProdRcpStep = 0 THEN
			//Mask Table
			tyP1040ProdSet.tyProdSet.tyStringSearch.uiMaskRtStat				:= FALSE;
			tyP1040ProdSet.tyProdSet.tyTableRecipe.uiMaskRtStat					:= FALSE;
			tyP1040ProdSet.tyProdSet.tyBtnDelete.uiMaskRtStat					:= FALSE;

			p_tyC0008MsgBox ACCESS ADR(tyP1040ProdSet.tyMsgBoxSaveAsk);

			IF tyP1040ProdSet.tyMsgBoxSaveAsk.tyBtnYes.bRtCompl = TRUE THEN
				tyP1040ProdSet.tyMsgBoxSaveAsk.tyBtnYes.bRtCompl				:= FALSE;
				tyP1040ProdSet.tyMsgBoxSaveAsk.tyBtnYes.bValue					:= FALSE;

				p_tyC0008MsgBox ACCESS ADR(tyP1040ProdSet.tyMsgBoxHide);

				usiSaveProdRcpStep	:= 1;

			ELSIF tyP1040ProdSet.tyMsgBoxSaveAsk.tyBtnNo.bRtCompl = TRUE THEN
				tyP1040ProdSet.tyMsgBoxSaveAsk.tyBtnNo.bRtCompl					:= FALSE;
				tyP1040ProdSet.tyMsgBoxSaveAsk.tyBtnNo.bValue					:= FALSE;

				p_tyC0008MsgBox ACCESS ADR(tyP1040ProdSet.tyMsgBoxHide);

				usiSaveProdRcpStep	:= 99;

			END_IF

		ELSIF usiSaveProdRcpStep = 1 THEN
			tyProdRcpInfoIn.sRcpNm			:= tyP1040ProdSet.tyProdSet.tyStringRecipeNm.sValue;
			tyProdRcpInfoIn.diWidthInUM		:= tyP1040ProdSet.tyProdSet.tyNumProdWidth.diValue;
			tyProdRcpInfoIn.diMaxSltValue	:= tyP1040ProdSet.tyProdSet.tyNumLastSlt.diValue;
			tyProdRcpInfoIn.diMinSltValue	:= tyP1040ProdSet.tyProdSet.tyNumFirstSlt.diValue;
			tyProdRcpInfoIn.diPitch			:= tyP1040ProdSet.tyProdSet.tyNumPitch.diValue;

			tyProdRcpInfoIn.usiMcMod		:= tyP1040ProdSet.tyProdSet.tyDrpDnMcMode.usiValueIdx;
			tyProdRcpInfoIn.usiFlippedBrd	:= tyP1040ProdSet.tyProdSet.tyDrpDnFlippedBrd.usiValueIdx;
			tyProdRcpInfoIn.bTopToBtm		:= p_tyNtParamCurr.bProjTopToBtmDefault;
			tyProdRcpInfoIn.bLongBrd		:= tyP1040ProdSet.tyProdSet.tyBtnLongBrd.bValue;

			tyProdRcpInfoIn.diPitchRear			:= tyP1040ProdSet.tyProdSet.tyNumPitchRear.diValue;
			tyProdRcpInfoIn.diWidthInUMRear		:= tyP1040ProdSet.tyProdSet.tyNumProdWidthRear.diValue;
			tyProdRcpInfoIn.diMaxSltValueRear	:= tyP1040ProdSet.tyProdSet.tyNumLastSltRear.diValue;
			tyProdRcpInfoIn.diMinSltValueRear	:= tyP1040ProdSet.tyProdSet.tyNumFirstSltRear.diValue;
			tyProdRcpInfoIn.diMtrPshrExtSpd		:= tyP1040ProdSet.tyProdSet.tyNumMtrPshrExtSpd.diValue;
			tyProdRcpInfoIn.diMtrPshrExtTorq	:= tyP1040ProdSet.tyProdSet.tyNumMtrPshrExtTorq.diValue;
			tyProdRcpInfoIn.diPshrOffset		:= tyP1040ProdSet.tyProdSet.tyNumPshrOffset.diValue;

			IF p_tyNtParamCurr.bLFProdWidth2Prep THEN
				tyProdRcpInfoIn.diWidthInUM2		:= tyP1040ProdSet.tyProdSet.tyNumProdWidth2.diValue;// ADD
			ELSE
				tyProdRcpInfoIn.diWidthInUM2		:= tyP1040ProdSet.tyProdSet.tyNumProdWidth.diValue;// ADD
			END_IF

			eProdRcpAct	:= ProdRcpActAddEdit;

			IF p_eProdRcpStat = ProdRcpActAddEdit AND p_eProdRcpStatus = Done THEN
				eProdRcpAct	:= ProdRcpActIdle;

				IF p_bProdRcpNmEmpty = TRUE THEN
					usiSaveProdRcpStep		:= 2;
				ELSIF p_bProdRcpListFull = TRUE THEN
					usiSaveProdRcpStep		:= 3;
				ELSE
					tyP1040ProdSet.tyProdSet.tyBtnSort.bValue := FALSE;
					tyP1040ProdSet.tyProdSet.tyStringSearch.sValue := '';

					bRefreshProdRcpTable	:= TRUE;
					bRefreshProdRcpDetail	:= TRUE;

					usiSaveProdRcpStep		:= 4;
				END_IF

			ELSIF p_eProdRcpStatus = Error THEN
				p_tyC0008MsgBox ACCESS ADR(tyP1040ProdSet.tyMsgBoxSaveErr);

				IF tyP1040ProdSet.tyMsgBoxSaveErr.tyBtnNo.bRtCompl = TRUE THEN
					tyP1040ProdSet.tyMsgBoxSaveErr.tyBtnNo.bRtCompl 			:= FALSE;
					tyP1040ProdSet.tyMsgBoxSaveErr.tyBtnNo.bValue 				:= FALSE;

					p_tyC0008MsgBox ACCESS ADR(tyP1040ProdSet.tyMsgBoxHide);

					usiSaveProdRcpStep		:= 99;
				END_IF
			END_IF

		// Product Recipe Param Error
		ELSIF usiSaveProdRcpStep = 2 THEN
			p_tyC0008MsgBox ACCESS ADR(tyP1040ProdSet.tyMsgBoxSaveNoNm);

			IF tyP1040ProdSet.tyMsgBoxSaveNoNm.tyBtnNo.bRtCompl = TRUE THEN
				tyP1040ProdSet.tyMsgBoxSaveNoNm.tyBtnNo.bRtCompl 				:= FALSE;
				tyP1040ProdSet.tyMsgBoxSaveNoNm.tyBtnNo.bValue 					:= FALSE;

				p_tyC0008MsgBox ACCESS ADR(tyP1040ProdSet.tyMsgBoxHide);

				usiSaveProdRcpStep		:= 99;
			END_IF

		// Prod Recipe List Full
		ELSIF usiSaveProdRcpStep = 3 THEN
			p_tyC0008MsgBox ACCESS ADR(tyP1040ProdSet.tyMsgBoxListFull);

			IF tyP1040ProdSet.tyMsgBoxListFull.tyBtnNo.bRtCompl = TRUE THEN
				tyP1040ProdSet.tyMsgBoxListFull.tyBtnNo.bRtCompl 				:= FALSE;
				tyP1040ProdSet.tyMsgBoxListFull.tyBtnNo.bValue 					:= FALSE;

				p_tyC0008MsgBox ACCESS ADR(tyP1040ProdSet.tyMsgBoxHide);

				usiSaveProdRcpStep		:= 99;
			END_IF

		ELSIF usiSaveProdRcpStep = 4 THEN
			IF tyProdRcpInfoIn.sRcpNm = p_tyProdRcpCurrRcp0.sRcpNm THEN
				p_tyC0008MsgBox ACCESS ADR(tyP1040ProdSet.tyMsgBoxReloadCurrRcp);

				IF tyP1040ProdSet.tyMsgBoxReloadCurrRcp.tyBtnNo.bRtCompl = TRUE THEN
					tyP1040ProdSet.tyMsgBoxReloadCurrRcp.tyBtnNo.bRtCompl 		:= FALSE;
					tyP1040ProdSet.tyMsgBoxReloadCurrRcp.tyBtnNo.bValue 		:= FALSE;

					p_tyC0008MsgBox ACCESS ADR(tyP1040ProdSet.tyMsgBoxHide);

					usiSaveProdRcpStep		:= 99;
				END_IF
			ELSE
				usiSaveProdRcpStep			:= 99;
			END_IF

		ELSIF usiSaveProdRcpStep = 99 THEN
			bRefreshProdRcpTable 			:= FALSE;

			//Unmask
			tyP1040ProdSet.tyProdSet.tyStringSearch.uiMaskRtStat	:= TRUE;
			tyP1040ProdSet.tyProdSet.tyTableRecipe.uiMaskRtStat		:= TRUE;
			tyP1040ProdSet.tyProdSet.tyBtnDelete.uiMaskRtStat		:= TRUE;

			//Reset
			tyP1040ProdSet.tyProdSet.tyBtnSave.bRtCompl	:= FALSE;
			tyP1040ProdSet.tyProdSet.tyBtnSave.bValue	:= FALSE;

			usiSaveProdRcpStep	:= 0;

		END_IF

	END_IF

END_ACTION
```

#### Act_OptP1050Keypad.st
```iecst
ACTION Act_OptP1050Keypad:

	IF fUIOutRtStatTPIsOpen(ADR(tyP1050LFSet.tyLdrEdit.tyStringIPAddr.uiRtStat)) THEN
		tyProperty.tyKeypad.tyStringTitle.sKeypadTitle	:= tyP1050LFSet.tyLdrEdit.tyStringIPAddr.sKeypadTitle;

	ELSIF fUIOutRtStatTPIsOpen(ADR(tyP1050LFSet.tyLdr.tyNumAfterOven.uiRtStat)) THEN
		tyProperty.tyKeypad.tyStringTitle.sKeypadTitle	:= tyP1050LFSet.tyLdr.tyNumAfterOven.sKeypadTitle;

	ELSIF fUIOutRtStatTPIsOpen(ADR(tyP1050LFSet.tyLdr.tyNumBeforeOven.uiRtStat)) THEN
		tyProperty.tyKeypad.tyStringTitle.sKeypadTitle	:= tyP1050LFSet.tyLdr.tyNumBeforeOven.sKeypadTitle;

	ELSIF fUIOutRtStatTPIsOpen(ADR(tyP1050LFSet.tyLdr.tyNumAfterOven2.uiRtStat)) THEN
		tyProperty.tyKeypad.tyStringTitle.sKeypadTitle	:= tyP1050LFSet.tyLdr.tyNumAfterOven2.sKeypadTitle;

	ELSIF fUIOutRtStatTPIsOpen(ADR(tyP1050LFSet.tyLdr.tyNumBeforeOven2.uiRtStat)) THEN
		tyProperty.tyKeypad.tyStringTitle.sKeypadTitle	:= tyP1050LFSet.tyLdr.tyNumBeforeOven2.sKeypadTitle;

	ELSE
		tyProperty.tyKeypad.tyStringTitle.sKeypadTitle	:= '';

	END_IF

END_ACTION
```

#### Act_OptP1050Table.st
```iecst
ACTION Act_OptP1050Table:

	//Call Table FB
	fbP1050Table.sVisuNm			:= tyP1050Table.sVisuNm;
	fbP1050Table.udiWorkAreaStartX	:= 96;
	fbP1050Table.udiWorkAreaEndX	:= 554;
	fbP1050Table.udiWorkAreaStartY	:= 75;
	fbP1050Table.udiWorkAreaEndY	:= 455;
	fbP1050Table.udiMinXDist		:= 20;
	fbP1050Table.udiMinYDist		:= 20;
	fbP1050Table.uiSlideScale		:= c_uiP1050TableSize;
	fbP1050Table.iTotalData			:= UDINT_TO_INT(c_diLFClntNum);
	fbP1050Table.iTotalRow			:= c_uiP1050TableSize;
	fbP1050Table(uiSliderStatus := tyP1050LFSet.tyLdr.tyTable1List.tyUISlider.uiRtStat , a_tyUIHotspot := tyP1050LFSet.tyLdr.tyTable1List.a_tyHotspot , uiTablePos := tyP1050Table.uiTablePos , iSliderPos := tyP1050LFSet.tyLdr.tyTable1List.tyUISlider.iValue);

	tyP1050Table.uiSelectedRow		:= fbP1050Table.uiSelectedRow;
	tyP1050Table.bTableActive		:= fbP1050Table.bTableActive;
	tyP1050Table.bSliderActive		:= fbP1050Table.bSliderActive;

	//Table Content
	IF tyP1050Table.bTableActive = TRUE OR tyP1050Table.bSliderActive = TRUE OR usiTableShftStep = 3 OR bUpdateP1050Table THEN
		FOR i := 1 TO c_uiP1050TableSize DO
			tyP1050LFSet.tyLdr.tyTable1List.a_tyStringDataCol0[i].sValue	:= UINT_TO_STRING(tyP1050Table.uiTablePos + i - 1);
			tyP1050LFSet.tyLdr.tyTable1List.a_tyStringDataCol2[i].sValue	:= p_tyMcParamCurr.a_sLFIPAddr[tyP1050Table.uiTablePos + i - 1];

			IF tyP1050LFSet.tyLdr.tyTable1List.a_tyStringDataCol2[i].sValue = '' THEN
				tyP1050LFSet.tyLdr.tyTable1List.a_tyTxtDataCol3[i].usiValueIdx	:= 0;
			ELSIF tyP1050LFSet.tyLdr.tyTable1List.a_tyStringDataCol2[i].sValue = '0000' THEN
				tyP1050LFSet.tyLdr.tyTable1List.a_tyTxtDataCol3[i].usiValueIdx	:= 3;
			ELSE
				tyP1050LFSet.tyLdr.tyTable1List.a_tyTxtDataCol3[i].usiValueIdx	:= (BOOL_TO_USINT(p_tyMcParamCurr.a_bLFOnline[tyP1050Table.uiTablePos + i - 1])) + 1;
			END_IF

		END_FOR

		IF bUpdateP1050Table THEN
			bUpdateP1050Table := FALSE;
		END_IF

	END_IF

	//Selected Row
	IF tyP1050Table.uiSelectedRow <> tyP1050Table.uiSelectedRowOld THEN

		FOR i := 1 TO c_uiP1050TableSize DO
			IF tyP1050Table.uiSelectedRow = i THEN
				tyP1050LFSet.tyLdr.tyTable1List.a_tyStringDataCol2[i].usiColor	:= 1;
				tyP1050LFSet.tyLdr.tyTable1List.a_tyTxtDataCol3[i].usiColor		:= 1;
			ELSE
				tyP1050LFSet.tyLdr.tyTable1List.a_tyStringDataCol2[i].usiColor	:= 0;
				tyP1050LFSet.tyLdr.tyTable1List.a_tyTxtDataCol3[i].usiColor		:= 0;
			END_IF
		END_FOR

		tyP1050Table.uiSelectedRowOld	:= tyP1050Table.uiSelectedRow;

	END_IF

END_ACTION
```

#### Act_OptP1080EditUsr.st
```iecst
ACTION Act_OptP1080EditUsr:

	// Edit User Display Control
	IF tyP1080UsrMgmt.tyUsrMgmt.tyBtnEditDetail.bRtCompl = TRUE THEN
		p_tyP1080UsrMgmtAct ACCESS ADR(tyP1080UsrMgmt.tyEdit);

		fUIInRtStatOff(ADR(tyP1080UsrMgmt.tyEdit.tyLyr.uiRtStat));
		fUIInRtStatHide(ADR(tyP1080UsrMgmt.tyUsrMgmt.tyLyr.uiRtStat));

		udiP1080SelectedRow		:= STRING_TO_UDINT(tyP1080UsrMgmt.tyUsrMgmt.tyTableList.a_tyStringDataCol0[tyP1080Table.uiSelectedRow].sValue);
		usiP1080SelectedLvl		:= tyP1080UsrMgmt.tyUsrMgmt.tyTableList.a_tyTxtDataCol3[tyP1080Table.uiSelectedRow].usiValueIdx;

		CASE tyP1080UsrMgmt.tyUsrMgmt.tyDrpDnLvl.usiValueIdx OF
			0:
				tyP1080UsrMgmt.tyEdit.tyStringUsrNm.sValue			:= p_tyUsrMgmtAllList[udiP1080SelectedRow].sUsrNm;
				tyP1080UsrMgmt.tyEdit.tyStringPw.sValue				:= p_tyUsrMgmtAllList[udiP1080SelectedRow].sPw;
				tyP1080UsrMgmt.tyEdit.tyDrpDnLvl.usiValueIdx		:= UDINT_TO_USINT((p_tyUsrMgmtAllList[udiP1080SelectedRow].eUsrLvl) - 1);

			1:
				tyP1080UsrMgmt.tyEdit.tyStringUsrNm.sValue			:= p_tyUsrMgmtLv2List[udiP1080SelectedRow].sUsrNm;
				tyP1080UsrMgmt.tyEdit.tyStringPw.sValue				:= p_tyUsrMgmtLv2List[udiP1080SelectedRow].sPw;
				tyP1080UsrMgmt.tyEdit.tyDrpDnLvl.usiValueIdx		:= UDINT_TO_USINT((p_tyUsrMgmtLv2List[udiP1080SelectedRow].eUsrLvl) - 1);

			2:
				tyP1080UsrMgmt.tyEdit.tyStringUsrNm.sValue			:= p_tyUsrMgmtLv3List[udiP1080SelectedRow].sUsrNm;
				tyP1080UsrMgmt.tyEdit.tyStringPw.sValue				:= p_tyUsrMgmtLv3List[udiP1080SelectedRow].sPw;
				tyP1080UsrMgmt.tyEdit.tyDrpDnLvl.usiValueIdx		:= UDINT_TO_USINT((p_tyUsrMgmtLv3List[udiP1080SelectedRow].eUsrLvl) - 1);

			3:
				tyP1080UsrMgmt.tyEdit.tyStringUsrNm.sValue			:= p_tyUsrMgmtAdminList[udiP1080SelectedRow].sUsrNm;
				tyP1080UsrMgmt.tyEdit.tyStringPw.sValue				:= p_tyUsrMgmtAdminList[udiP1080SelectedRow].sPw;
				tyP1080UsrMgmt.tyEdit.tyDrpDnLvl.usiValueIdx		:= UDINT_TO_USINT((p_tyUsrMgmtAdminList[udiP1080SelectedRow].eUsrLvl) - 1);
		END_CASE

		tyP1080UsrMgmt.tyEdit.tyStringPw.sValue						:= '';

		IF usiP1080SelectedLvl = 5 OR usiP1080SelectedLvl = 6 THEN
			tyP1080UsrMgmt.tyEdit.tyDrpDnLvl.usiValueMinIdx			:= 3;
			tyP1080UsrMgmt.tyEdit.tyDrpDnLvl.usiValueMaxIdx			:= 4;
		ELSE
			tyP1080UsrMgmt.tyEdit.tyDrpDnLvl.usiValueMinIdx			:= 0;
			tyP1080UsrMgmt.tyEdit.tyDrpDnLvl.usiValueMaxIdx			:= 2;
		END_IF

		tyP1080UsrMgmt.tyUsrMgmt.tyBtnEditDetail.bRtCompl			:= FALSE;
		tyP1080UsrMgmt.tyUsrMgmt.tyBtnEditDetail.bValue				:= TRUE;

	END_IF

	// Edit User
	IF tyP1080UsrMgmt.tyUsrMgmt.tyBtnEditDetail.bValue = TRUE THEN
		IF tyP1080UsrMgmt.tyEdit.tyBtnOk.bRtCompl = TRUE THEN
			IF usiEditUsrMgmtStep = 0 THEN
				tyUsrMgmtInfoIn.sUsrNm			:= tyP1080UsrMgmt.tyEdit.tyStringUsrNm.sValue;
				tyUsrMgmtInfoIn.sPw				:= tyP1080UsrMgmt.tyEdit.tyStringPw.sValue;
				tyUsrMgmtInfoIn.eUsrLvl			:= tyP1080UsrMgmt.tyEdit.tyDrpDnLvl.usiValueIdx + 1;

				eUsrMgmtAct					:= UsrMgmtActEdit;

				IF p_eUsrMgmtStat = UsrMgmtActEdit AND p_eUsrMgmtStatus = Done THEN
					eUsrMgmtAct				:= UsrMgmtActIdle;

					IF p_bUsrMgmtNmEmpty = TRUE THEN
						usiEditUsrMgmtStep		:= 1;
					ELSIF p_bUsrMgmtListFull = TRUE THEN
						usiEditUsrMgmtStep		:= 2;
					ELSE
						bRefreshUsrMgmtTable	:= TRUE;
						usiEditUsrMgmtStep		:= 99;
					END_IF
				ELSIF p_eUsrMgmtStatus = Error THEN
					p_tyC0008MsgBox ACCESS ADR(tyP1080UsrMgmt.tyMsgBoxEditErr);

					IF tyP1080UsrMgmt.tyMsgBoxEditErr.tyBtnNo.bRtCompl = TRUE THEN
						tyP1080UsrMgmt.tyMsgBoxEditErr.tyBtnNo.bRtCompl 		:= FALSE;
						tyP1080UsrMgmt.tyMsgBoxEditErr.tyBtnNo.bValue 			:= FALSE;

						p_tyC0008MsgBox ACCESS ADR(tyP1080UsrMgmt.tyMsgBoxHide);

						usiEditUsrMgmtStep		:= 99;
					END_IF
				END_IF

			// User Managment Param Invalid
			ELSIF usiEditUsrMgmtStep = 1 THEN
				p_tyC0008MsgBox ACCESS ADR(tyP1080UsrMgmt.tyMsgBoxEditParamErr);

				IF tyP1080UsrMgmt.tyMsgBoxEditParamErr.tyBtnNo.bRtCompl = TRUE THEN
					tyP1080UsrMgmt.tyMsgBoxEditParamErr.tyBtnNo.bRtCompl 		:= FALSE;
					tyP1080UsrMgmt.tyMsgBoxEditParamErr.tyBtnNo.bValue 			:= FALSE;

					p_tyC0008MsgBox ACCESS ADR(tyP1040ProdSet.tyMsgBoxHide);

					tyP1080UsrMgmt.tyEdit.tyStringPw.sValue						:= '';
					tyP1080UsrMgmt.tyEdit.tyDrpDnLvl.usiValueIdx				:= 0;

					tyP1080UsrMgmt.tyEdit.tyBtnOk.bRtCompl 						:= FALSE;
					tyP1080UsrMgmt.tyEdit.tyBtnOk.bValue 						:= FALSE;

					usiEditUsrMgmtStep			:= 0;
				END_IF

			// User Managment List Full
			ELSIF usiEditUsrMgmtStep = 2 THEN
				p_tyC0008MsgBox ACCESS ADR(tyP1080UsrMgmt.tyMsgBoxListFull);

				IF tyP1080UsrMgmt.tyMsgBoxListFull.tyBtnNo.bRtCompl = TRUE THEN
					tyP1080UsrMgmt.tyMsgBoxListFull.tyBtnNo.bRtCompl 			:= FALSE;
					tyP1080UsrMgmt.tyMsgBoxListFull.tyBtnNo.bValue 				:= FALSE;

					p_tyC0008MsgBox ACCESS ADR(tyP1080UsrMgmt.tyMsgBoxHide);

					usiEditUsrMgmtStep			:= 99;
				END_IF

			ELSIF usiEditUsrMgmtStep = 99 THEN
				fUIInRtStatOff(ADR(tyP1080UsrMgmt.tyUsrMgmt.tyLyr.uiRtStat));
				fUIInRtStatHide(ADR(tyP1080UsrMgmt.tyEdit.tyLyr.uiRtStat));

				tyP1080UsrMgmt.tyUsrMgmt.tyBtnEditDetail.bValue					:= FALSE;

				tyP1080UsrMgmt.tyEdit.tyBtnOk.bRtCompl							:= FALSE;
				tyP1080UsrMgmt.tyEdit.tyBtnOk.bValue							:= FALSE;

				usiEditUsrMgmtStep				:= 0;
			END_IF

		ELSIF tyP1080UsrMgmt.tyEdit.tyBtnCancel.bRtCompl = TRUE THEN
			fUIInRtStatOff(ADR(tyP1080UsrMgmt.tyUsrMgmt.tyLyr.uiRtStat));
			fUIInRtStatHide(ADR(tyP1080UsrMgmt.tyEdit.tyLyr.uiRtStat));

			tyP1080UsrMgmt.tyUsrMgmt.tyBtnEditDetail.bValue						:= FALSE;

			tyP1080UsrMgmt.tyEdit.tyBtnCancel.bRtCompl							:= FALSE;
			tyP1080UsrMgmt.tyEdit.tyBtnCancel.bValue							:= FALSE;
		END_IF
	END_IF

END_ACTION
```

#### Act_EntP1081Disp.st
```iecst
ACTION Act_EntP1081Disp:

	// Access
	p_tyC0004Navi ACCESS ADR(tyP1081UsrMgmtUsrAccessRgt.tyNaviBack);

	p_tyC0005Main ACCESS ADR(tyCommon.tyMain);

	p_tyC0006Set ACCESS ADR(tyCommon.tySet);

	p_tyC0007Notif ACCESS ADR(tyCommon.tyNotif);

	p_tyC0008MsgBox ACCESS ADR(tyP1081UsrMgmtUsrAccessRgt.tyMsgBoxHide);

	p_tyC0009Info ACCESS ADR(tyCommon.tyInfo);

	p_tyP1081UsrMgmtUsrAccessRgtSel ACCESS ADR(tyP1081UsrMgmtUsrAccessRgt.tyUsrAccessRgtSel);
	p_tyP1081UsrMgmtUsrAccessRgt ACCESS ADR(tyP1081UsrMgmtUsrAccessRgt.tyUsrAccessRgtLvl1);

	// Reset DrpDn List
	tyP1081UsrMgmtUsrAccessRgt.tyUsrAccessRgtSel.tyDrpDnLevel.usiValueIdx			:= 0;

	//Backup Param
	tyP1081UsrMgmtUsrAccessRgt.tyUsrAccessRgtLvl1BkUp			:= tyP1081UsrMgmtUsrAccessRgt.tyUsrAccessRgtLvl1;
	tyP1081UsrMgmtUsrAccessRgt.tyUsrAccessRgtLvl2BkUp			:= tyP1081UsrMgmtUsrAccessRgt.tyUsrAccessRgtLvl2;
	tyP1081UsrMgmtUsrAccessRgt.tyUsrAccessRgtLvl3BkUp			:= tyP1081UsrMgmtUsrAccessRgt.tyUsrAccessRgtLvl3;

END_ACTION
```

#### Act_OptP1081Save.st
```iecst
ACTION Act_OptP1081Save:

	// Level 1
	IF tyP1081UsrMgmtUsrAccessRgt.tyUsrAccessRgtLvl1.tyStringNm.bRtCompl 					OR tyP1081UsrMgmtUsrAccessRgt.tyUsrAccessRgtLvl1.tyBtnOps.bRtCompl
		OR tyP1081UsrMgmtUsrAccessRgt.tyUsrAccessRgtLvl1.tyBtnProdSel.bRtCompl				OR tyP1081UsrMgmtUsrAccessRgt.tyUsrAccessRgtLvl1.tyBtnMagSel.bRtCompl
		OR tyP1081UsrMgmtUsrAccessRgt.tyUsrAccessRgtLvl1.tyBtnMcInfo.bRtCompl				OR tyP1081UsrMgmtUsrAccessRgt.tyUsrAccessRgtLvl1.tyBtnAlm.bRtCompl
		OR tyP1081UsrMgmtUsrAccessRgt.tyUsrAccessRgtLvl1.tyBtnBffrInfo.bRtCompl				OR tyP1081UsrMgmtUsrAccessRgt.tyUsrAccessRgtLvl1.tyBtnOvenInfo.bRtCompl
		OR tyP1081UsrMgmtUsrAccessRgt.tyUsrAccessRgtLvl1.tyBtnMagInfo.bRtCompl				OR tyP1081UsrMgmtUsrAccessRgt.tyUsrAccessRgtLvl1.tyBtnLFCtrl.bRtCompl
		OR tyP1081UsrMgmtUsrAccessRgt.tyUsrAccessRgtLvl1.tyBtnManual.bRtCompl				OR tyP1081UsrMgmtUsrAccessRgt.tyUsrAccessRgtLvl1.tyBtnSimu.bRtCompl
		OR tyP1081UsrMgmtUsrAccessRgt.tyUsrAccessRgtLvl1.tyBtnProdSet.bRtCompl				OR tyP1081UsrMgmtUsrAccessRgt.tyUsrAccessRgtLvl1.tyBtnMagSet.bRtCompl
		OR tyP1081UsrMgmtUsrAccessRgt.tyUsrAccessRgtLvl1.tyBtnMcSet.bRtCompl				OR tyP1081UsrMgmtUsrAccessRgt.tyUsrAccessRgtLvl1.tyBtnLang.bRtCompl
		OR tyP1081UsrMgmtUsrAccessRgt.tyUsrAccessRgtLvl1.tyBtnLFSet.bRtCompl				OR tyP1081UsrMgmtUsrAccessRgt.tyUsrAccessRgtLvl1.tyBtnChgParam.bRtCompl
		OR tyP1081UsrMgmtUsrAccessRgt.tyUsrAccessRgtLvl1.tyBtnManualFBOnly.bRtCompl

		// Level 2
		OR tyP1081UsrMgmtUsrAccessRgt.tyUsrAccessRgtLvl2.tyStringNm.bRtCompl 				OR tyP1081UsrMgmtUsrAccessRgt.tyUsrAccessRgtLvl2.tyBtnOps.bRtCompl
		OR tyP1081UsrMgmtUsrAccessRgt.tyUsrAccessRgtLvl2.tyBtnProdSel.bRtCompl				OR tyP1081UsrMgmtUsrAccessRgt.tyUsrAccessRgtLvl2.tyBtnMagSel.bRtCompl
		OR tyP1081UsrMgmtUsrAccessRgt.tyUsrAccessRgtLvl2.tyBtnMcInfo.bRtCompl				OR tyP1081UsrMgmtUsrAccessRgt.tyUsrAccessRgtLvl2.tyBtnAlm.bRtCompl
		OR tyP1081UsrMgmtUsrAccessRgt.tyUsrAccessRgtLvl2.tyBtnBffrInfo.bRtCompl				OR tyP1081UsrMgmtUsrAccessRgt.tyUsrAccessRgtLvl2.tyBtnOvenInfo.bRtCompl
		OR tyP1081UsrMgmtUsrAccessRgt.tyUsrAccessRgtLvl2.tyBtnMagInfo.bRtCompl				OR tyP1081UsrMgmtUsrAccessRgt.tyUsrAccessRgtLvl2.tyBtnLFCtrl.bRtCompl
		OR tyP1081UsrMgmtUsrAccessRgt.tyUsrAccessRgtLvl2.tyBtnManual.bRtCompl				OR tyP1081UsrMgmtUsrAccessRgt.tyUsrAccessRgtLvl2.tyBtnSimu.bRtCompl
		OR tyP1081UsrMgmtUsrAccessRgt.tyUsrAccessRgtLvl2.tyBtnProdSet.bRtCompl				OR tyP1081UsrMgmtUsrAccessRgt.tyUsrAccessRgtLvl2.tyBtnMagSet.bRtCompl
		OR tyP1081UsrMgmtUsrAccessRgt.tyUsrAccessRgtLvl2.tyBtnMcSet.bRtCompl				OR tyP1081UsrMgmtUsrAccessRgt.tyUsrAccessRgtLvl2.tyBtnLang.bRtCompl
		OR tyP1081UsrMgmtUsrAccessRgt.tyUsrAccessRgtLvl2.tyBtnLFSet.bRtCompl				OR tyP1081UsrMgmtUsrAccessRgt.tyUsrAccessRgtLvl2.tyBtnChgParam.bRtCompl
		OR tyP1081UsrMgmtUsrAccessRgt.tyUsrAccessRgtLvl2.tyBtnManualFBOnly.bRtCompl

		// Level 3
		OR tyP1081UsrMgmtUsrAccessRgt.tyUsrAccessRgtLvl3.tyStringNm.bRtCompl 				OR tyP1081UsrMgmtUsrAccessRgt.tyUsrAccessRgtLvl3.tyBtnOps.bRtCompl
		OR tyP1081UsrMgmtUsrAccessRgt.tyUsrAccessRgtLvl3.tyBtnProdSel.bRtCompl				OR tyP1081UsrMgmtUsrAccessRgt.tyUsrAccessRgtLvl3.tyBtnMagSel.bRtCompl
		OR tyP1081UsrMgmtUsrAccessRgt.tyUsrAccessRgtLvl3.tyBtnMcInfo.bRtCompl				OR tyP1081UsrMgmtUsrAccessRgt.tyUsrAccessRgtLvl3.tyBtnAlm.bRtCompl
		OR tyP1081UsrMgmtUsrAccessRgt.tyUsrAccessRgtLvl3.tyBtnBffrInfo.bRtCompl				OR tyP1081UsrMgmtUsrAccessRgt.tyUsrAccessRgtLvl3.tyBtnOvenInfo.bRtCompl
		OR tyP1081UsrMgmtUsrAccessRgt.tyUsrAccessRgtLvl3.tyBtnMagInfo.bRtCompl				OR tyP1081UsrMgmtUsrAccessRgt.tyUsrAccessRgtLvl3.tyBtnLFCtrl.bRtCompl
		OR tyP1081UsrMgmtUsrAccessRgt.tyUsrAccessRgtLvl3.tyBtnManual.bRtCompl				OR tyP1081UsrMgmtUsrAccessRgt.tyUsrAccessRgtLvl3.tyBtnSimu.bRtCompl
		OR tyP1081UsrMgmtUsrAccessRgt.tyUsrAccessRgtLvl3.tyBtnProdSet.bRtCompl				OR tyP1081UsrMgmtUsrAccessRgt.tyUsrAccessRgtLvl3.tyBtnMagSet.bRtCompl
		OR tyP1081UsrMgmtUsrAccessRgt.tyUsrAccessRgtLvl3.tyBtnMcSet.bRtCompl				OR tyP1081UsrMgmtUsrAccessRgt.tyUsrAccessRgtLvl3.tyBtnLang.bRtCompl
		OR tyP1081UsrMgmtUsrAccessRgt.tyUsrAccessRgtLvl3.tyBtnLFSet.bRtCompl				OR tyP1081UsrMgmtUsrAccessRgt.tyUsrAccessRgtLvl3.tyBtnChgParam.bRtCompl
		OR tyP1081UsrMgmtUsrAccessRgt.tyUsrAccessRgtLvl3.tyBtnManualFBOnly.bRtCompl THEN

		fUIInRtStatHide(ADR(tyCommon.tySet.tyBtnSave.uiMaskRtStat));

		// Level 1
		tyP1081UsrMgmtUsrAccessRgt.tyUsrAccessRgtLvl1.tyStringNm.bRtCompl 		:= FALSE;
		tyP1081UsrMgmtUsrAccessRgt.tyUsrAccessRgtLvl1.tyBtnOps.bRtCompl 		:= FALSE;
		tyP1081UsrMgmtUsrAccessRgt.tyUsrAccessRgtLvl1.tyBtnProdSel.bRtCompl 	:= FALSE;
		tyP1081UsrMgmtUsrAccessRgt.tyUsrAccessRgtLvl1.tyBtnMagSel.bRtCompl 		:= FALSE;
		tyP1081UsrMgmtUsrAccessRgt.tyUsrAccessRgtLvl1.tyBtnMcInfo.bRtCompl		:= FALSE;
		tyP1081UsrMgmtUsrAccessRgt.tyUsrAccessRgtLvl1.tyBtnAlm.bRtCompl			:= FALSE;
		tyP1081UsrMgmtUsrAccessRgt.tyUsrAccessRgtLvl1.tyBtnBffrInfo.bRtCompl	:= FALSE;
		tyP1081UsrMgmtUsrAccessRgt.tyUsrAccessRgtLvl1.tyBtnOvenInfo.bRtCompl	:= FALSE;
		tyP1081UsrMgmtUsrAccessRgt.tyUsrAccessRgtLvl1.tyBtnMagInfo.bRtCompl		:= FALSE;
		tyP1081UsrMgmtUsrAccessRgt.tyUsrAccessRgtLvl1.tyBtnLFCtrl.bRtCompl		:= FALSE;
		tyP1081UsrMgmtUsrAccessRgt.tyUsrAccessRgtLvl1.tyBtnManual.bRtCompl		:= FALSE;
		tyP1081UsrMgmtUsrAccessRgt.tyUsrAccessRgtLvl1.tyBtnSimu.bRtCompl		:= FALSE;
		tyP1081UsrMgmtUsrAccessRgt.tyUsrAccessRgtLvl1.tyBtnProdSet.bRtCompl		:= FALSE;
		tyP1081UsrMgmtUsrAccessRgt.tyUsrAccessRgtLvl1.tyBtnMagSet.bRtCompl		:= FALSE;
		tyP1081UsrMgmtUsrAccessRgt.tyUsrAccessRgtLvl1.tyBtnMcSet.bRtCompl		:= FALSE;
		tyP1081UsrMgmtUsrAccessRgt.tyUsrAccessRgtLvl1.tyBtnLang.bRtCompl		:= FALSE;
		tyP1081UsrMgmtUsrAccessRgt.tyUsrAccessRgtLvl1.tyBtnLFSet.bRtCompl		:= FALSE;
		tyP1081UsrMgmtUsrAccessRgt.tyUsrAccessRgtLvl1.tyBtnChgParam.bRtCompl	:= FALSE;
		tyP1081UsrMgmtUsrAccessRgt.tyUsrAccessRgtLvl1.tyBtnManualFBOnly.bRtCompl:= FALSE;

		// Level 2
		tyP1081UsrMgmtUsrAccessRgt.tyUsrAccessRgtLvl2.tyStringNm.bRtCompl 		:= FALSE;
		tyP1081UsrMgmtUsrAccessRgt.tyUsrAccessRgtLvl2.tyBtnOps.bRtCompl 		:= FALSE;
		tyP1081UsrMgmtUsrAccessRgt.tyUsrAccessRgtLvl2.tyBtnProdSel.bRtCompl 	:= FALSE;
		tyP1081UsrMgmtUsrAccessRgt.tyUsrAccessRgtLvl2.tyBtnMagSel.bRtCompl 		:= FALSE;
		tyP1081UsrMgmtUsrAccessRgt.tyUsrAccessRgtLvl2.tyBtnMcInfo.bRtCompl		:= FALSE;
		tyP1081UsrMgmtUsrAccessRgt.tyUsrAccessRgtLvl2.tyBtnAlm.bRtCompl			:= FALSE;
		tyP1081UsrMgmtUsrAccessRgt.tyUsrAccessRgtLvl2.tyBtnBffrInfo.bRtCompl	:= FALSE;
		tyP1081UsrMgmtUsrAccessRgt.tyUsrAccessRgtLvl2.tyBtnOvenInfo.bRtCompl	:= FALSE;
		tyP1081UsrMgmtUsrAccessRgt.tyUsrAccessRgtLvl2.tyBtnMagInfo.bRtCompl		:= FALSE;
		tyP1081UsrMgmtUsrAccessRgt.tyUsrAccessRgtLvl2.tyBtnLFCtrl.bRtCompl		:= FALSE;
		tyP1081UsrMgmtUsrAccessRgt.tyUsrAccessRgtLvl2.tyBtnManual.bRtCompl		:= FALSE;
		tyP1081UsrMgmtUsrAccessRgt.tyUsrAccessRgtLvl2.tyBtnSimu.bRtCompl		:= FALSE;
		tyP1081UsrMgmtUsrAccessRgt.tyUsrAccessRgtLvl2.tyBtnProdSet.bRtCompl		:= FALSE;
		tyP1081UsrMgmtUsrAccessRgt.tyUsrAccessRgtLvl2.tyBtnMagSet.bRtCompl		:= FALSE;
		tyP1081UsrMgmtUsrAccessRgt.tyUsrAccessRgtLvl2.tyBtnMcSet.bRtCompl		:= FALSE;
		tyP1081UsrMgmtUsrAccessRgt.tyUsrAccessRgtLvl2.tyBtnLang.bRtCompl		:= FALSE;
		tyP1081UsrMgmtUsrAccessRgt.tyUsrAccessRgtLvl2.tyBtnLFSet.bRtCompl		:= FALSE;
		tyP1081UsrMgmtUsrAccessRgt.tyUsrAccessRgtLvl2.tyBtnChgParam.bRtCompl	:= FALSE;
		tyP1081UsrMgmtUsrAccessRgt.tyUsrAccessRgtLvl2.tyBtnManualFBOnly.bRtCompl:= FALSE;

		// Level 3
		tyP1081UsrMgmtUsrAccessRgt.tyUsrAccessRgtLvl3.tyStringNm.bRtCompl 		:= FALSE;
		tyP1081UsrMgmtUsrAccessRgt.tyUsrAccessRgtLvl3.tyBtnOps.bRtCompl 		:= FALSE;
		tyP1081UsrMgmtUsrAccessRgt.tyUsrAccessRgtLvl3.tyBtnProdSel.bRtCompl 	:= FALSE;
		tyP1081UsrMgmtUsrAccessRgt.tyUsrAccessRgtLvl3.tyBtnMagSel.bRtCompl 		:= FALSE;
		tyP1081UsrMgmtUsrAccessRgt.tyUsrAccessRgtLvl3.tyBtnMcInfo.bRtCompl		:= FALSE;
		tyP1081UsrMgmtUsrAccessRgt.tyUsrAccessRgtLvl3.tyBtnAlm.bRtCompl			:= FALSE;
		tyP1081UsrMgmtUsrAccessRgt.tyUsrAccessRgtLvl3.tyBtnBffrInfo.bRtCompl	:= FALSE;
		tyP1081UsrMgmtUsrAccessRgt.tyUsrAccessRgtLvl3.tyBtnOvenInfo.bRtCompl	:= FALSE;
		tyP1081UsrMgmtUsrAccessRgt.tyUsrAccessRgtLvl3.tyBtnMagInfo.bRtCompl		:= FALSE;
		tyP1081UsrMgmtUsrAccessRgt.tyUsrAccessRgtLvl3.tyBtnLFCtrl.bRtCompl		:= FALSE;
		tyP1081UsrMgmtUsrAccessRgt.tyUsrAccessRgtLvl3.tyBtnManual.bRtCompl		:= FALSE;
		tyP1081UsrMgmtUsrAccessRgt.tyUsrAccessRgtLvl3.tyBtnSimu.bRtCompl		:= FALSE;
		tyP1081UsrMgmtUsrAccessRgt.tyUsrAccessRgtLvl3.tyBtnProdSet.bRtCompl		:= FALSE;
		tyP1081UsrMgmtUsrAccessRgt.tyUsrAccessRgtLvl3.tyBtnMagSet.bRtCompl		:= FALSE;
		tyP1081UsrMgmtUsrAccessRgt.tyUsrAccessRgtLvl3.tyBtnMcSet.bRtCompl		:= FALSE;
		tyP1081UsrMgmtUsrAccessRgt.tyUsrAccessRgtLvl3.tyBtnLang.bRtCompl		:= FALSE;
		tyP1081UsrMgmtUsrAccessRgt.tyUsrAccessRgtLvl3.tyBtnLFSet.bRtCompl		:= FALSE;
		tyP1081UsrMgmtUsrAccessRgt.tyUsrAccessRgtLvl3.tyBtnChgParam.bRtCompl	:= FALSE;
		tyP1081UsrMgmtUsrAccessRgt.tyUsrAccessRgtLvl3.tyBtnManualFBOnly.bRtCompl:= FALSE;

	END_IF

	IF tyCommon.tySet.tyBtnSave.bRtCompl = TRUE THEN
		//Save Param
		CASE tyP1081UsrMgmtUsrAccessRgt.tyUsrAccessRgtSel.tyDrpDnLevel.usiValueIdx OF
			0:
				tyUsrMgmtAccessRightLvl1Wr.sNm					:= tyP1081UsrMgmtUsrAccessRgt.tyUsrAccessRgtLvl1.tyStringNm.sValue;
				tyUsrMgmtAccessRightLvl1Wr.bOpt					:= tyP1081UsrMgmtUsrAccessRgt.tyUsrAccessRgtLvl1.tyBtnOps.bValue;
				tyUsrMgmtAccessRightLvl1Wr.bProdSel				:= tyP1081UsrMgmtUsrAccessRgt.tyUsrAccessRgtLvl1.tyBtnProdSel.bValue;
				tyUsrMgmtAccessRightLvl1Wr.bMagSel				:= tyP1081UsrMgmtUsrAccessRgt.tyUsrAccessRgtLvl1.tyBtnMagSel.bValue;
				tyUsrMgmtAccessRightLvl1Wr.bMcInfo				:= tyP1081UsrMgmtUsrAccessRgt.tyUsrAccessRgtLvl1.tyBtnMcInfo.bValue;
				tyUsrMgmtAccessRightLvl1Wr.bAlm					:= tyP1081UsrMgmtUsrAccessRgt.tyUsrAccessRgtLvl1.tyBtnAlm.bValue;
				tyUsrMgmtAccessRightLvl1Wr.bBffrInfo			:= tyP1081UsrMgmtUsrAccessRgt.tyUsrAccessRgtLvl1.tyBtnBffrInfo.bValue;
				tyUsrMgmtAccessRightLvl1Wr.bOvenInfo			:= tyP1081UsrMgmtUsrAccessRgt.tyUsrAccessRgtLvl1.tyBtnOvenInfo.bValue;
				tyUsrMgmtAccessRightLvl1Wr.bMagInfo				:= tyP1081UsrMgmtUsrAccessRgt.tyUsrAccessRgtLvl1.tyBtnMagInfo.bValue;
				tyUsrMgmtAccessRightLvl1Wr.bLFCtrl				:= tyP1081UsrMgmtUsrAccessRgt.tyUsrAccessRgtLvl1.tyBtnLFCtrl.bValue;
				tyUsrMgmtAccessRightLvl1Wr.bManual				:= tyP1081UsrMgmtUsrAccessRgt.tyUsrAccessRgtLvl1.tyBtnManual.bValue;
				tyUsrMgmtAccessRightLvl1Wr.bSimulation			:= tyP1081UsrMgmtUsrAccessRgt.tyUsrAccessRgtLvl1.tyBtnSimu.bValue;
				tyUsrMgmtAccessRightLvl1Wr.bProdSet				:= tyP1081UsrMgmtUsrAccessRgt.tyUsrAccessRgtLvl1.tyBtnProdSet.bValue;
				tyUsrMgmtAccessRightLvl1Wr.bMagSet				:= tyP1081UsrMgmtUsrAccessRgt.tyUsrAccessRgtLvl1.tyBtnMagSet.bValue;
				tyUsrMgmtAccessRightLvl1Wr.bMcSet				:= tyP1081UsrMgmtUsrAccessRgt.tyUsrAccessRgtLvl1.tyBtnMcSet.bValue;
				tyUsrMgmtAccessRightLvl1Wr.bLang				:= tyP1081UsrMgmtUsrAccessRgt.tyUsrAccessRgtLvl1.tyBtnLang.bValue;
				tyUsrMgmtAccessRightLvl1Wr.bLFSet				:= tyP1081UsrMgmtUsrAccessRgt.tyUsrAccessRgtLvl1.tyBtnLFSet.bValue;
				tyUsrMgmtAccessRightLvl1Wr.bChgParam			:= tyP1081UsrMgmtUsrAccessRgt.tyUsrAccessRgtLvl1.tyBtnChgParam.bValue;
				tyUsrMgmtAccessRightLvl1Wr.bManualFBOnly		:= tyP1081UsrMgmtUsrAccessRgt.tyUsrAccessRgtLvl1.tyBtnManualFBOnly.bValue;

			1:
				tyUsrMgmtAccessRightLvl2Wr.sNm					:= tyP1081UsrMgmtUsrAccessRgt.tyUsrAccessRgtLvl2.tyStringNm.sValue;
				tyUsrMgmtAccessRightLvl2Wr.bOpt					:= tyP1081UsrMgmtUsrAccessRgt.tyUsrAccessRgtLvl2.tyBtnOps.bValue;
				tyUsrMgmtAccessRightLvl2Wr.bProdSel				:= tyP1081UsrMgmtUsrAccessRgt.tyUsrAccessRgtLvl2.tyBtnProdSel.bValue;
				tyUsrMgmtAccessRightLvl2Wr.bMagSel				:= tyP1081UsrMgmtUsrAccessRgt.tyUsrAccessRgtLvl2.tyBtnMagSel.bValue;
				tyUsrMgmtAccessRightLvl2Wr.bMcInfo				:= tyP1081UsrMgmtUsrAccessRgt.tyUsrAccessRgtLvl2.tyBtnMcInfo.bValue;
				tyUsrMgmtAccessRightLvl2Wr.bAlm					:= tyP1081UsrMgmtUsrAccessRgt.tyUsrAccessRgtLvl2.tyBtnAlm.bValue;
				tyUsrMgmtAccessRightLvl2Wr.bBffrInfo			:= tyP1081UsrMgmtUsrAccessRgt.tyUsrAccessRgtLvl2.tyBtnBffrInfo.bValue;
				tyUsrMgmtAccessRightLvl2Wr.bOvenInfo			:= tyP1081UsrMgmtUsrAccessRgt.tyUsrAccessRgtLvl2.tyBtnOvenInfo.bValue;
				tyUsrMgmtAccessRightLvl2Wr.bMagInfo				:= tyP1081UsrMgmtUsrAccessRgt.tyUsrAccessRgtLvl2.tyBtnMagInfo.bValue;
				tyUsrMgmtAccessRightLvl2Wr.bLFCtrl				:= tyP1081UsrMgmtUsrAccessRgt.tyUsrAccessRgtLvl2.tyBtnLFCtrl.bValue;
				tyUsrMgmtAccessRightLvl2Wr.bManual				:= tyP1081UsrMgmtUsrAccessRgt.tyUsrAccessRgtLvl2.tyBtnManual.bValue;
				tyUsrMgmtAccessRightLvl2Wr.bSimulation			:= tyP1081UsrMgmtUsrAccessRgt.tyUsrAccessRgtLvl2.tyBtnSimu.bValue;
				tyUsrMgmtAccessRightLvl2Wr.bProdSet				:= tyP1081UsrMgmtUsrAccessRgt.tyUsrAccessRgtLvl2.tyBtnProdSet.bValue;
				tyUsrMgmtAccessRightLvl2Wr.bMagSet				:= tyP1081UsrMgmtUsrAccessRgt.tyUsrAccessRgtLvl2.tyBtnMagSet.bValue;
				tyUsrMgmtAccessRightLvl2Wr.bMcSet				:= tyP1081UsrMgmtUsrAccessRgt.tyUsrAccessRgtLvl2.tyBtnMcSet.bValue;
				tyUsrMgmtAccessRightLvl2Wr.bLang				:= tyP1081UsrMgmtUsrAccessRgt.tyUsrAccessRgtLvl2.tyBtnLang.bValue;
				tyUsrMgmtAccessRightLvl2Wr.bLFSet				:= tyP1081UsrMgmtUsrAccessRgt.tyUsrAccessRgtLvl2.tyBtnLFSet.bValue;
				tyUsrMgmtAccessRightLvl2Wr.bChgParam			:= tyP1081UsrMgmtUsrAccessRgt.tyUsrAccessRgtLvl2.tyBtnChgParam.bValue;
				tyUsrMgmtAccessRightLvl2Wr.bManualFBOnly		:= tyP1081UsrMgmtUsrAccessRgt.tyUsrAccessRgtLvl2.tyBtnManualFBOnly.bValue;

			2:
				tyUsrMgmtAccessRightLvl3Wr.sNm					:= tyP1081UsrMgmtUsrAccessRgt.tyUsrAccessRgtLvl3.tyStringNm.sValue;
				tyUsrMgmtAccessRightLvl3Wr.bOpt					:= tyP1081UsrMgmtUsrAccessRgt.tyUsrAccessRgtLvl3.tyBtnOps.bValue;
				tyUsrMgmtAccessRightLvl3Wr.bProdSel				:= tyP1081UsrMgmtUsrAccessRgt.tyUsrAccessRgtLvl3.tyBtnProdSel.bValue;
				tyUsrMgmtAccessRightLvl3Wr.bMagSel				:= tyP1081UsrMgmtUsrAccessRgt.tyUsrAccessRgtLvl3.tyBtnMagSel.bValue;
				tyUsrMgmtAccessRightLvl3Wr.bMcInfo				:= tyP1081UsrMgmtUsrAccessRgt.tyUsrAccessRgtLvl3.tyBtnMcInfo.bValue;
				tyUsrMgmtAccessRightLvl3Wr.bAlm					:= tyP1081UsrMgmtUsrAccessRgt.tyUsrAccessRgtLvl3.tyBtnAlm.bValue;
				tyUsrMgmtAccessRightLvl3Wr.bBffrInfo			:= tyP1081UsrMgmtUsrAccessRgt.tyUsrAccessRgtLvl3.tyBtnBffrInfo.bValue;
				tyUsrMgmtAccessRightLvl3Wr.bOvenInfo			:= tyP1081UsrMgmtUsrAccessRgt.tyUsrAccessRgtLvl3.tyBtnOvenInfo.bValue;
				tyUsrMgmtAccessRightLvl3Wr.bMagInfo				:= tyP1081UsrMgmtUsrAccessRgt.tyUsrAccessRgtLvl3.tyBtnMagInfo.bValue;
				tyUsrMgmtAccessRightLvl3Wr.bLFCtrl				:= tyP1081UsrMgmtUsrAccessRgt.tyUsrAccessRgtLvl3.tyBtnLFCtrl.bValue;
				tyUsrMgmtAccessRightLvl3Wr.bManual				:= tyP1081UsrMgmtUsrAccessRgt.tyUsrAccessRgtLvl3.tyBtnManual.bValue;
				tyUsrMgmtAccessRightLvl3Wr.bSimulation			:= tyP1081UsrMgmtUsrAccessRgt.tyUsrAccessRgtLvl3.tyBtnSimu.bValue;
				tyUsrMgmtAccessRightLvl3Wr.bProdSet				:= tyP1081UsrMgmtUsrAccessRgt.tyUsrAccessRgtLvl3.tyBtnProdSet.bValue;
				tyUsrMgmtAccessRightLvl3Wr.bMagSet				:= tyP1081UsrMgmtUsrAccessRgt.tyUsrAccessRgtLvl3.tyBtnMagSet.bValue;
				tyUsrMgmtAccessRightLvl3Wr.bMcSet				:= tyP1081UsrMgmtUsrAccessRgt.tyUsrAccessRgtLvl3.tyBtnMcSet.bValue;
				tyUsrMgmtAccessRightLvl3Wr.bLang				:= tyP1081UsrMgmtUsrAccessRgt.tyUsrAccessRgtLvl3.tyBtnLang.bValue;
				tyUsrMgmtAccessRightLvl3Wr.bLFSet				:= tyP1081UsrMgmtUsrAccessRgt.tyUsrAccessRgtLvl3.tyBtnLFSet.bValue;
				tyUsrMgmtAccessRightLvl3Wr.bChgParam			:= tyP1081UsrMgmtUsrAccessRgt.tyUsrAccessRgtLvl3.tyBtnChgParam.bValue;
				tyUsrMgmtAccessRightLvl3Wr.bManualFBOnly		:= tyP1081UsrMgmtUsrAccessRgt.tyUsrAccessRgtLvl3.tyBtnManualFBOnly.bValue;
		END_CASE

		eUsrMgmtAct	:= UsrMgmtActSaveAccessRight;

		IF p_eUsrMgmtStat = UsrMgmtActSaveAccessRight AND p_eUsrMgmtStatus = Done THEN
			eUsrMgmtAct	:= UsrMgmtActIdle;

			//Backup Param
			tyP1081UsrMgmtUsrAccessRgt.tyUsrAccessRgtLvl1BkUp		:= tyP1081UsrMgmtUsrAccessRgt.tyUsrAccessRgtLvl1;
			tyP1081UsrMgmtUsrAccessRgt.tyUsrAccessRgtLvl2BkUp		:= tyP1081UsrMgmtUsrAccessRgt.tyUsrAccessRgtLvl2;
			tyP1081UsrMgmtUsrAccessRgt.tyUsrAccessRgtLvl3BkUp		:= tyP1081UsrMgmtUsrAccessRgt.tyUsrAccessRgtLvl3;

			CASE tyP1081UsrMgmtUsrAccessRgt.tyUsrAccessRgtSel.tyDrpDnLevel.usiValueIdx OF
				0:
					tyProperty.tyUITxtSnippets.sUsrMgmtUsrLv1Nm		:= tyP1081UsrMgmtUsrAccessRgt.tyUsrAccessRgtLvl1.tyStringNm.sValue;
				1:
					tyProperty.tyUITxtSnippets.sUsrMgmtUsrLv2Nm		:= tyP1081UsrMgmtUsrAccessRgt.tyUsrAccessRgtLvl2.tyStringNm.sValue;
				2:
					tyProperty.tyUITxtSnippets.sUsrMgmtUsrLv3Nm		:= tyP1081UsrMgmtUsrAccessRgt.tyUsrAccessRgtLvl3.tyStringNm.sValue;
			END_CASE

			tyCommon.tySet.tyBtnSave.bRtCompl						:= FALSE;

			fUIInRtStatOff(ADR(tyCommon.tySet.tyBtnSave.uiMaskRtStat));

		ELSIF p_eUsrMgmtStatus = Error THEN
			p_tyC0008MsgBox ACCESS ADR(tyP1081UsrMgmtUsrAccessRgt.tyMsgBoxSaveErr);

			IF tyP1081UsrMgmtUsrAccessRgt.tyMsgBoxSaveErr.tyBtnNo.bRtCompl = TRUE THEN
				tyP1081UsrMgmtUsrAccessRgt.tyMsgBoxSaveErr.tyBtnNo.bRtCompl 				:= FALSE;
				tyP1081UsrMgmtUsrAccessRgt.tyMsgBoxSaveErr.tyBtnNo.bValue 					:= FALSE;

				p_tyC0008MsgBox ACCESS ADR(tyP1081UsrMgmtUsrAccessRgt.tyMsgBoxHide);

				//Recover Param
				tyUsrMgmtAccessRightLvl1Wr	:= p_tyUsrMgmtFullData.tyAccessRightLvl1;
				tyUsrMgmtAccessRightLvl2Wr	:= p_tyUsrMgmtFullData.tyAccessRightLvl2;
				tyUsrMgmtAccessRightLvl3Wr	:= p_tyUsrMgmtFullData.tyAccessRightLvl3;

				tyP1081UsrMgmtUsrAccessRgt.tyUsrAccessRgtLvl1	:= tyP1081UsrMgmtUsrAccessRgt.tyUsrAccessRgtLvl1BkUp;
				tyP1081UsrMgmtUsrAccessRgt.tyUsrAccessRgtLvl2	:= tyP1081UsrMgmtUsrAccessRgt.tyUsrAccessRgtLvl2BkUp;
				tyP1081UsrMgmtUsrAccessRgt.tyUsrAccessRgtLvl3	:= tyP1081UsrMgmtUsrAccessRgt.tyUsrAccessRgtLvl3BkUp;

				tyCommon.tySet.tyBtnSave.bRtCompl	:= FALSE;
				fUIInRtStatOff(ADR(tyCommon.tySet.tyBtnSave.uiMaskRtStat));
			END_IF
		END_IF
	END_IF

END_ACTION
```

#### Program Logical/UI/UI/Act_Background/Action/P0003

##### Act_EntP0003Disp.st
```iecst
ACTION Act_EntP0003Disp:

	//Access
	p_tyC0005Main ACCESS ADR(tyCommon.tyMain1);

	p_tyC0007Notif ACCESS ADR(tyCommon.tyNotif);

	p_tyP0003Gen ACCESS ADR(tyP0003MMenu.tyMMenuGen);

	IF NOT bPromptSessionExp THEN
		p_tyC0008MsgBox ACCESS ADR(tyP0003MMenu.tyMsgBoxHide);
	END_IF

	p_tyC0009Info ACCESS ADR(tyCommon.tyInfo);

	p_tyP0003BtnAuto ACCESS ADR(tyP0003MMenu.tyMMenuBtn.tyBtnAuto);
	p_tyP0003BtnStop ACCESS ADR(tyP0003MMenu.tyMMenuBtn.tyBtnStop);
	p_tyP0003BtnReset ACCESS ADR(tyP0003MMenu.tyMMenuBtn.tyBtnReset);
	p_tyP0003BtnBuz ACCESS ADR(tyP0003MMenu.tyMMenuBtn.tyBtnBuz);
	p_tyP0003AcceptData ACCESS ADR(tyP0003MMenu.tyMMenuBtn.tyBtnAccDat);

	tyP0003MMenu.tyMMenuBtn.tyBtnBuz.uiRtStat.0 := NOT (p_tyNtParamCurr.tyDOSettings.diBuzzer > 0);

	//{TextSnippet_1} Position in Main Menu

	//hide corresponding button
//	tyP0003MMenu.tyMMenuBtn.tyBtnUnload.uiRtStat.0 :=  NOT p_tyNtParamCurr.bProjLifterMagPlatform;
	tyP0003MMenu.tyMMenuBtn.tyBtnRlsNewMag1.uiRtStat.0 := p_tyMcParamCurr.eMagExMode = McSetMagXcAutoMode AND p_tyMcParamCurr.eAGVComProtocol <> McSetAGVCommDisabled OR p_tyNtParamCurr.bProjLifterMagPlatform;
	tyP0003MMenu.tyMMenuBtn.tyBtnRlsNewMag2.uiRtStat.0 := p_tyMcParamCurr.eMagExMode = McSetMagXcAutoMode AND p_tyMcParamCurr.eAGVComProtocol <> McSetAGVCommDisabled OR p_tyNtParamCurr.bProjLifterMagPlatform;
	tyP0003MMenu.tyMMenuBtn.tyBtnRlsNewMag3.uiRtStat.0 := p_tyMcParamCurr.eMagExMode = McSetMagXcAutoMode AND p_tyMcParamCurr.eAGVComProtocol <> McSetAGVCommDisabled OR p_tyNtParamCurr.bProjLifterMagPlatform;

	//idx =1 start from
	usiPosidx := 1 ;
	FOR usidx:= 1 TO SIZEOF(p_tyMcParamCurr.aButtonPos)/SIZEOF(p_tyMcParamCurr.aButtonPos[1]) DO
		IF NOT(p_tyNtParamCurr.tyDOSettings.diBuzzer > 0 AND usidx = 1)THEN

			//p_eCurrBtnPos ACCESS (ADR(p_tyMcParamCurr.tyOptBtnPos) + usiPosidx*SIZEOF(p_tyMcParamCurr.tyOptBtnPos.ePos1));

			IF p_tyMcParamCurr.aButtonPos[usiPosidx] = eNA THEN
				a_tyPtrtoAddr[usidx] :=   ADR(tyP0003MMenu.tyMMenuBtn.tyBtnHide);
			ELSIF p_tyMcParamCurr.aButtonPos[usiPosidx] = eMnlUnload THEN
				a_tyPtrtoAddr[usidx] :=   ADR(tyP0003MMenu.tyMMenuBtn.tyBtnUnload);
			ELSIF p_tyMcParamCurr.aButtonPos[usiPosidx]= eRlsNewMag1 THEN
				a_tyPtrtoAddr[usidx] :=   ADR(tyP0003MMenu.tyMMenuBtn.tyBtnRlsNewMag1);
			ELSIF p_tyMcParamCurr.aButtonPos[usiPosidx]= eRlsNewMag2 THEN
				a_tyPtrtoAddr[usidx] :=   ADR(tyP0003MMenu.tyMMenuBtn.tyBtnRlsNewMag2);
			ELSIF p_tyMcParamCurr.aButtonPos[usiPosidx] = eRlsNewMag3 THEN
				a_tyPtrtoAddr[usidx] :=   ADR(tyP0003MMenu.tyMMenuBtn.tyBtnRlsNewMag3);
			END_IF
			usiPosidx := usiPosidx +1;
		ELSE
			a_tyPtrtoAddr[usidx] :=   ADR(tyP0003MMenu.tyMMenuBtn.tyBtnHide);
		END_IF
	END_FOR
	p_tyP0003Btn1 ACCESS a_tyPtrtoAddr[1];
	p_tyP0003Btn2 ACCESS a_tyPtrtoAddr[2];
	p_tyP0003Btn3 ACCESS a_tyPtrtoAddr[3];
	p_tyP0003Btn4 ACCESS a_tyPtrtoAddr[4];
	p_tyP0003Btn5 ACCESS a_tyPtrtoAddr[5];
	p_tyP0003Btn6 ACCESS a_tyPtrtoAddr[6];
	p_tyP0003Btn7 ACCESS a_tyPtrtoAddr[7];

	//Not Used
//	p_tyP0003Btn4 ACCESS ADR(tyP0003MMenu.tyMMenuBtn.tyBtn4);// If not used, hide it in the data type
//	p_tyP0003Btn5 ACCESS ADR(tyP0003MMenu.tyMMenuBtn.tyBtn5);// If not used, hide it in the data type
//	p_tyP0003Btn6 ACCESS ADR(tyP0003MMenu.tyMMenuBtn.tyBtn6);// If not used, hide it in the data type
//	p_tyP0003Btn7 ACCESS ADR(tyP0003MMenu.tyMMenuBtn.tyBtn7);// If not used, hide it in the data type

END_ACTION
```

##### Act_OptP0003UpdtStat.st
```iecst
ACTION Act_OptP0003UpdtStat:

	IF p_bOpsStatusRun THEN
		tyP0003MMenu.tyMMenuGen.tyStatusTxt.usiValueIdx := 20;
	ELSIF p_bOpsStatusCycleStop THEN
		tyP0003MMenu.tyMMenuGen.tyStatusTxt.usiValueIdx := 21;
	ELSIF p_bAlarmErr THEN
		tyP0003MMenu.tyMMenuGen.tyStatusTxt.usiValueIdx := 22;
	ELSE
		tyP0003MMenu.tyMMenuGen.tyStatusTxt.usiValueIdx := 23;
	END_IF

	//SMEMA Indicator
	IF p_tyNtParamCurr.bUIConvDirRL = FALSE THEN
		fUIInRtStatHide(ADR(tyP0003MMenu.tyMMenuGen.tyBitmapDSAComm1.uiMaskRtStat));
		fUIInRtStatHide(ADR(tyP0003MMenu.tyMMenuGen.tyBitmapDSBComm1.uiMaskRtStat));
		IF p_tyMcParamCurr.eDSCommA = McSetCommModSMEMA THEN
			fUIInRtStatHide(ADR(tyP0003MMenu.tyMMenuGen.tyBitmapDSAComm.uiMaskRtStat));
		ELSIF p_tyMcParamCurr.eDSCommA = McSetCommModHermes THEN
			IF p_bDSHermesAConnected = TRUE THEN
				fUIInRtStatHide(ADR(tyP0003MMenu.tyMMenuGen.tyBitmapDSAComm.uiMaskRtStat));
			ELSE
				fUIInRtStatOff(ADR(tyP0003MMenu.tyMMenuGen.tyBitmapDSAComm.uiMaskRtStat));
			END_IF
		END_IF

		IF p_tyMcParamCurr.eDSCommB = McSetCommModSMEMA THEN
			fUIInRtStatHide(ADR(tyP0003MMenu.tyMMenuGen.tyBitmapDSBComm.uiMaskRtStat));
		ELSIF p_tyMcParamCurr.eDSCommB = McSetCommModHermes THEN
			IF p_bDSHermesBConnected = TRUE THEN
				fUIInRtStatHide(ADR(tyP0003MMenu.tyMMenuGen.tyBitmapDSBComm.uiMaskRtStat));
			ELSE
				fUIInRtStatOff(ADR(tyP0003MMenu.tyMMenuGen.tyBitmapDSBComm.uiMaskRtStat));
			END_IF
		END_IF
	ELSE
		fUIInRtStatHide(ADR(tyP0003MMenu.tyMMenuGen.tyBitmapDSAComm.uiMaskRtStat));
		fUIInRtStatHide(ADR(tyP0003MMenu.tyMMenuGen.tyBitmapDSBComm.uiMaskRtStat));
		IF p_tyMcParamCurr.eDSCommA = McSetCommModSMEMA THEN
			fUIInRtStatHide(ADR(tyP0003MMenu.tyMMenuGen.tyBitmapDSAComm1.uiMaskRtStat));
		ELSIF p_tyMcParamCurr.eDSCommA = McSetCommModHermes THEN
			IF p_bDSHermesAConnected = TRUE THEN
				fUIInRtStatHide(ADR(tyP0003MMenu.tyMMenuGen.tyBitmapDSAComm1.uiMaskRtStat));
			ELSE
				fUIInRtStatOff(ADR(tyP0003MMenu.tyMMenuGen.tyBitmapDSAComm1.uiMaskRtStat));
			END_IF
		END_IF

		IF p_tyMcParamCurr.eDSCommB = McSetCommModSMEMA THEN
			fUIInRtStatHide(ADR(tyP0003MMenu.tyMMenuGen.tyBitmapDSBComm1.uiMaskRtStat));
		ELSIF p_tyMcParamCurr.eDSCommB = McSetCommModHermes THEN
			IF p_bDSHermesBConnected = TRUE THEN
				fUIInRtStatHide(ADR(tyP0003MMenu.tyMMenuGen.tyBitmapDSBComm1.uiMaskRtStat));
			ELSE
				fUIInRtStatOff(ADR(tyP0003MMenu.tyMMenuGen.tyBitmapDSBComm1.uiMaskRtStat));
			END_IF
		END_IF
	END_IF

	//Communication - Signal
	//DBA A
	IF p_tyNtParamCurr.bUIConvDirRL = FALSE THEN
		IF p_tyMcParamCurr.eDSCommA = McSetCommModSMEMA THEN
			IF p_bDSSMEMAAUSRdy = TRUE THEN
				IF p_bDSSMEMAAUSGdBrdRdy = TRUE THEN
					tyP0003MMenu.tyMMenuGen.tyBitmapDSOut.usiValueIdx	:= 1;
				ELSE
					tyP0003MMenu.tyMMenuGen.tyBitmapDSOut.usiValueIdx	:= 2;
				END_IF
			ELSE
				tyP0003MMenu.tyMMenuGen.tyBitmapDSOut.usiValueIdx	:= 0;
			END_IF

		ELSIF p_tyMcParamCurr.eDSCommA = McSetCommModHermes THEN
			IF p_bDSHermesAUSRdy = TRUE THEN
				IF p_bDSHermesAUSGdRdy = TRUE THEN
					tyP0003MMenu.tyMMenuGen.tyBitmapDSOut.usiValueIdx	:= 1;
				ELSE
					tyP0003MMenu.tyMMenuGen.tyBitmapDSOut.usiValueIdx	:= 2;
				END_IF
			ELSE
				tyP0003MMenu.tyMMenuGen.tyBitmapDSOut.usiValueIdx	:= 0;
			END_IF

		END_IF
	ELSE
		IF p_tyMcParamCurr.eDSCommA = McSetCommModSMEMA THEN
			IF p_bDSSMEMAAUSRdy = TRUE THEN
				IF p_bDSSMEMAAUSGdBrdRdy = TRUE THEN
					tyP0003MMenu.tyMMenuGen.tyBitmapDSOut1.usiValueIdx	:= 1;
				ELSE
					tyP0003MMenu.tyMMenuGen.tyBitmapDSOut1.usiValueIdx	:= 2;
				END_IF
			ELSE
				tyP0003MMenu.tyMMenuGen.tyBitmapDSOut1.usiValueIdx	:= 0;
			END_IF

		ELSIF p_tyMcParamCurr.eDSCommA = McSetCommModHermes THEN
			IF p_bDSHermesAUSRdy = TRUE THEN
				IF p_bDSHermesAUSGdRdy = TRUE THEN
					tyP0003MMenu.tyMMenuGen.tyBitmapDSOut1.usiValueIdx	:= 1;
				ELSE
					tyP0003MMenu.tyMMenuGen.tyBitmapDSOut1.usiValueIdx	:= 2;
				END_IF
			ELSE
				tyP0003MMenu.tyMMenuGen.tyBitmapDSOut1.usiValueIdx	:= 0;
			END_IF

		END_IF
	END_IF

	//DSB A
	IF p_tyNtParamCurr.bUIConvDirRL = FALSE THEN
		IF p_tyMcParamCurr.eDSCommA = McSetCommModSMEMA THEN
			IF p_bDSSMEMAADSRdy = TRUE THEN
				tyP0003MMenu.tyMMenuGen.tyBitmapDSIn.usiValueIdx	:= 1;
			ELSE
				tyP0003MMenu.tyMMenuGen.tyBitmapDSIn.usiValueIdx	:= 0;
			END_IF

		ELSIF p_tyMcParamCurr.eDSCommA = McSetCommModHermes THEN
			IF p_bDSHermesADSRdy = TRUE THEN
				IF p_bDSHermesADSGdRdy = TRUE THEN
					tyP0003MMenu.tyMMenuGen.tyBitmapDSIn.usiValueIdx	:= 1;
				ELSE
					tyP0003MMenu.tyMMenuGen.tyBitmapDSIn.usiValueIdx	:= 2;
				END_IF
			ELSE
				tyP0003MMenu.tyMMenuGen.tyBitmapDSIn.usiValueIdx	:= 0;
			END_IF

		END_IF
	ELSE
		IF p_tyMcParamCurr.eDSCommA = McSetCommModSMEMA THEN
			IF p_bDSSMEMAADSRdy = TRUE THEN
				tyP0003MMenu.tyMMenuGen.tyBitmapDSIn1.usiValueIdx	:= 1;
			ELSE
				tyP0003MMenu.tyMMenuGen.tyBitmapDSIn1.usiValueIdx	:= 0;
			END_IF

		ELSIF p_tyMcParamCurr.eDSCommA = McSetCommModHermes THEN
			IF p_bDSHermesADSRdy = TRUE THEN
				IF p_bDSHermesADSGdRdy = TRUE THEN
					tyP0003MMenu.tyMMenuGen.tyBitmapDSIn1.usiValueIdx	:= 1;
				ELSE
					tyP0003MMenu.tyMMenuGen.tyBitmapDSIn1.usiValueIdx	:= 2;
				END_IF
			ELSE
				tyP0003MMenu.tyMMenuGen.tyBitmapDSIn1.usiValueIdx	:= 0;
			END_IF

		END_IF
	END_IF
	//DBA B
	IF p_tyNtParamCurr.bUIConvDirRL = FALSE THEN
		IF p_tyMcParamCurr.eDSCommB = McSetCommModSMEMA THEN
			IF p_bDSSMEMABUSRdy = TRUE THEN
				IF p_bDSSMEMABUSGdBrdRdy = TRUE THEN
					tyP0003MMenu.tyMMenuGen.tyBitmapDSBOut.usiValueIdx	:= 1;
				ELSE
					tyP0003MMenu.tyMMenuGen.tyBitmapDSBOut.usiValueIdx	:= 2;
				END_IF
			ELSE
				tyP0003MMenu.tyMMenuGen.tyBitmapDSBOut.usiValueIdx	:= 0;
			END_IF

		ELSIF p_tyMcParamCurr.eDSCommB = McSetCommModHermes THEN
			IF p_bDSHermesBUSRdy = TRUE THEN
				IF p_bDSHermesBUSGdRdy = TRUE THEN
					tyP0003MMenu.tyMMenuGen.tyBitmapDSBOut.usiValueIdx	:= 1;
				ELSE
					tyP0003MMenu.tyMMenuGen.tyBitmapDSBOut.usiValueIdx	:= 2;
				END_IF
			ELSE
				tyP0003MMenu.tyMMenuGen.tyBitmapDSBOut.usiValueIdx	:= 0;
			END_IF

		END_IF
	ELSE
		IF p_tyMcParamCurr.eDSCommB = McSetCommModSMEMA THEN
			IF p_bDSSMEMABUSRdy = TRUE THEN
				IF p_bDSSMEMABUSGdBrdRdy = TRUE THEN
					tyP0003MMenu.tyMMenuGen.tyBitmapDSBOut1.usiValueIdx	:= 1;
				ELSE
					tyP0003MMenu.tyMMenuGen.tyBitmapDSBOut1.usiValueIdx	:= 2;
				END_IF
			ELSE
				tyP0003MMenu.tyMMenuGen.tyBitmapDSBOut1.usiValueIdx	:= 0;
			END_IF

		ELSIF p_tyMcParamCurr.eDSCommB = McSetCommModHermes THEN
			IF p_bDSHermesBUSRdy = TRUE THEN
				IF p_bDSHermesBUSGdRdy = TRUE THEN
					tyP0003MMenu.tyMMenuGen.tyBitmapDSBOut1.usiValueIdx	:= 1;
				ELSE
					tyP0003MMenu.tyMMenuGen.tyBitmapDSBOut1.usiValueIdx	:= 2;
				END_IF
			ELSE
				tyP0003MMenu.tyMMenuGen.tyBitmapDSBOut1.usiValueIdx	:= 0;
			END_IF

		END_IF
	END_IF

	//DSB B
	IF p_tyNtParamCurr.bUIConvDirRL = FALSE THEN
		IF p_tyMcParamCurr.eDSCommB = McSetCommModSMEMA THEN
			IF p_bDSSMEMABDSRdy = TRUE THEN
				tyP0003MMenu.tyMMenuGen.tyBitmapDSBIn.usiValueIdx	:= 1;
			ELSE
				tyP0003MMenu.tyMMenuGen.tyBitmapDSBIn.usiValueIdx	:= 0;
			END_IF

		ELSIF p_tyMcParamCurr.eDSCommB = McSetCommModHermes THEN
			IF p_bDSHermesBDSRdy = TRUE THEN
				IF p_bDSHermesBDSGdRdy = TRUE THEN
					tyP0003MMenu.tyMMenuGen.tyBitmapDSBIn.usiValueIdx	:= 1;
				ELSE
					tyP0003MMenu.tyMMenuGen.tyBitmapDSBIn.usiValueIdx	:= 2;
				END_IF
			ELSE
				tyP0003MMenu.tyMMenuGen.tyBitmapDSBIn.usiValueIdx	:= 0;
			END_IF

		END_IF
	ELSE
		IF p_tyMcParamCurr.eDSCommB = McSetCommModSMEMA THEN
			IF p_bDSSMEMABDSRdy = TRUE THEN
				tyP0003MMenu.tyMMenuGen.tyBitmapDSBIn1.usiValueIdx	:= 1;
			ELSE
				tyP0003MMenu.tyMMenuGen.tyBitmapDSBIn1.usiValueIdx	:= 0;
			END_IF

		ELSIF p_tyMcParamCurr.eDSCommB = McSetCommModHermes THEN
			IF p_bDSHermesBDSRdy = TRUE THEN
				IF p_bDSHermesBDSGdRdy = TRUE THEN
					tyP0003MMenu.tyMMenuGen.tyBitmapDSBIn1.usiValueIdx	:= 1;
				ELSE
					tyP0003MMenu.tyMMenuGen.tyBitmapDSBIn1.usiValueIdx	:= 2;
				END_IF
			ELSE
				tyP0003MMenu.tyMMenuGen.tyBitmapDSBIn1.usiValueIdx	:= 0;
			END_IF

		END_IF
	END_IF

	//Current last zone product recipe name

	tyP0003MMenu.tyMMenuGen.tyStringProdNm.sValue := p_tyProdRcpCurrRcp1.sRcpNm;

END_ACTION
```

#### Program Logical/UI/UI/Act_Background/Action/P1024

##### Act_OptP1024Keypad.st
```iecst
ACTION Act_OptP1024Keypad:

	IF fUIOutRtStatTPIsOpen(ADR(tyP1024McSetAntiGap.tyAntiGap.tyNumLftSenOff.uiRtStat)) = TRUE THEN
		tyProperty.tyKeypad.tyStringTitle.sKeypadTitle	:= tyP1024McSetAntiGap.tyAntiGap.tyNumLftSenOff.sKeypadTitle;

	ELSIF fUIOutRtStatTPIsOpen(ADR(tyP1024McSetAntiGap.tyAntiGap.tyNumRgtSenOff.uiRtStat)) = TRUE THEN
		tyProperty.tyKeypad.tyStringTitle.sKeypadTitle	:= tyP1024McSetAntiGap.tyAntiGap.tyNumRgtSenOff.sKeypadTitle;

	ELSIF fUIOutRtStatTPIsOpen(ADR(tyP1024McSetAntiGap.tyAntiGap.tyNumMagConvEntOff.uiRtStat)) = TRUE THEN
		tyProperty.tyKeypad.tyStringTitle.sKeypadTitle	:= tyP1024McSetAntiGap.tyAntiGap.tyNumMagConvEntOff.sKeypadTitle;

	ELSIF fUIOutRtStatTPIsOpen(ADR(tyP1024McSetAntiGap.tyAntiGap.tyNumMagConvEntOn.uiRtStat)) = TRUE THEN
		tyProperty.tyKeypad.tyStringTitle.sKeypadTitle	:= tyP1024McSetAntiGap.tyAntiGap.tyNumMagConvEntOn.sKeypadTitle;

	ELSIF fUIOutRtStatTPIsOpen(ADR(tyP1024McSetAntiGap.tyAntiGap.tyNumMagConvPresentOff.uiRtStat)) = TRUE THEN
		tyProperty.tyKeypad.tyStringTitle.sKeypadTitle	:= tyP1024McSetAntiGap.tyAntiGap.tyNumMagConvEntOn.sKeypadTitle;

	ELSIF fUIOutRtStatTPIsOpen(ADR(tyP1024McSetAntiGap.tyAntiGap.tyNumMagConvPresentOn.uiRtStat)) = TRUE THEN
		tyProperty.tyKeypad.tyStringTitle.sKeypadTitle	:= tyP1024McSetAntiGap.tyAntiGap.tyNumMagConvEntOn.sKeypadTitle;
	END_IF

END_ACTION
```
